      AN    OV;
      =     L      0.0;
      A     L      0.0;
      A(    ;
      A     M   1014.1;
      A(    ;
      A     I   1010.3;
      A(    ;
      ON    I     68.7;
      ON    I     69.4;
      )     ;
      O     ;
      A     I   1018.2;
      A(    ;
      ON    I     68.3;
      ON    I     69.2;
      )     ;
      )     ;
      O     ;
      A     M   1014.0;
      A(    ;
      O     I   1018.2;
      O     ;
      A     I   1018.3;
      A     M    284.0;
      A     M   4710.0;
      )     ;
      A(    ;
      ON    I     71.3;
      ON    I     71.4;
      )     ;
      )     ;
      =     L      0.1;
      A     L      0.1;
      A     T     12;
      S     M   1003.2;
      A     L      0.1;
      AN    M   1004.0;
      AN    M   1004.1;
      AN    M   6060.1;
      AN    M   6260.0;
      AN    M   6280.0;
      AN    M   1004.2;
      L     S5T#500MS;
      SD    T     12;
      A     L      0.0;
      A     I      0.1;
      A(    ;
      A     M   1014.1;
      A(    ;
      A     I     68.7;
      A     I     69.4;
      A     I     68.3;
      A     I     69.2;
      O     ;
      AN    M   1001.4;
      A     M   1001.6;
      A     I     68.3;
      A     I     69.2;
      )     ;
      O     ;
      A     M   1014.0;
      A     M   1001.6;
      A     I     71.3;
      A     I     71.4;
      )     ;
      R     M   1003.2;
NETWORK
TITLE =
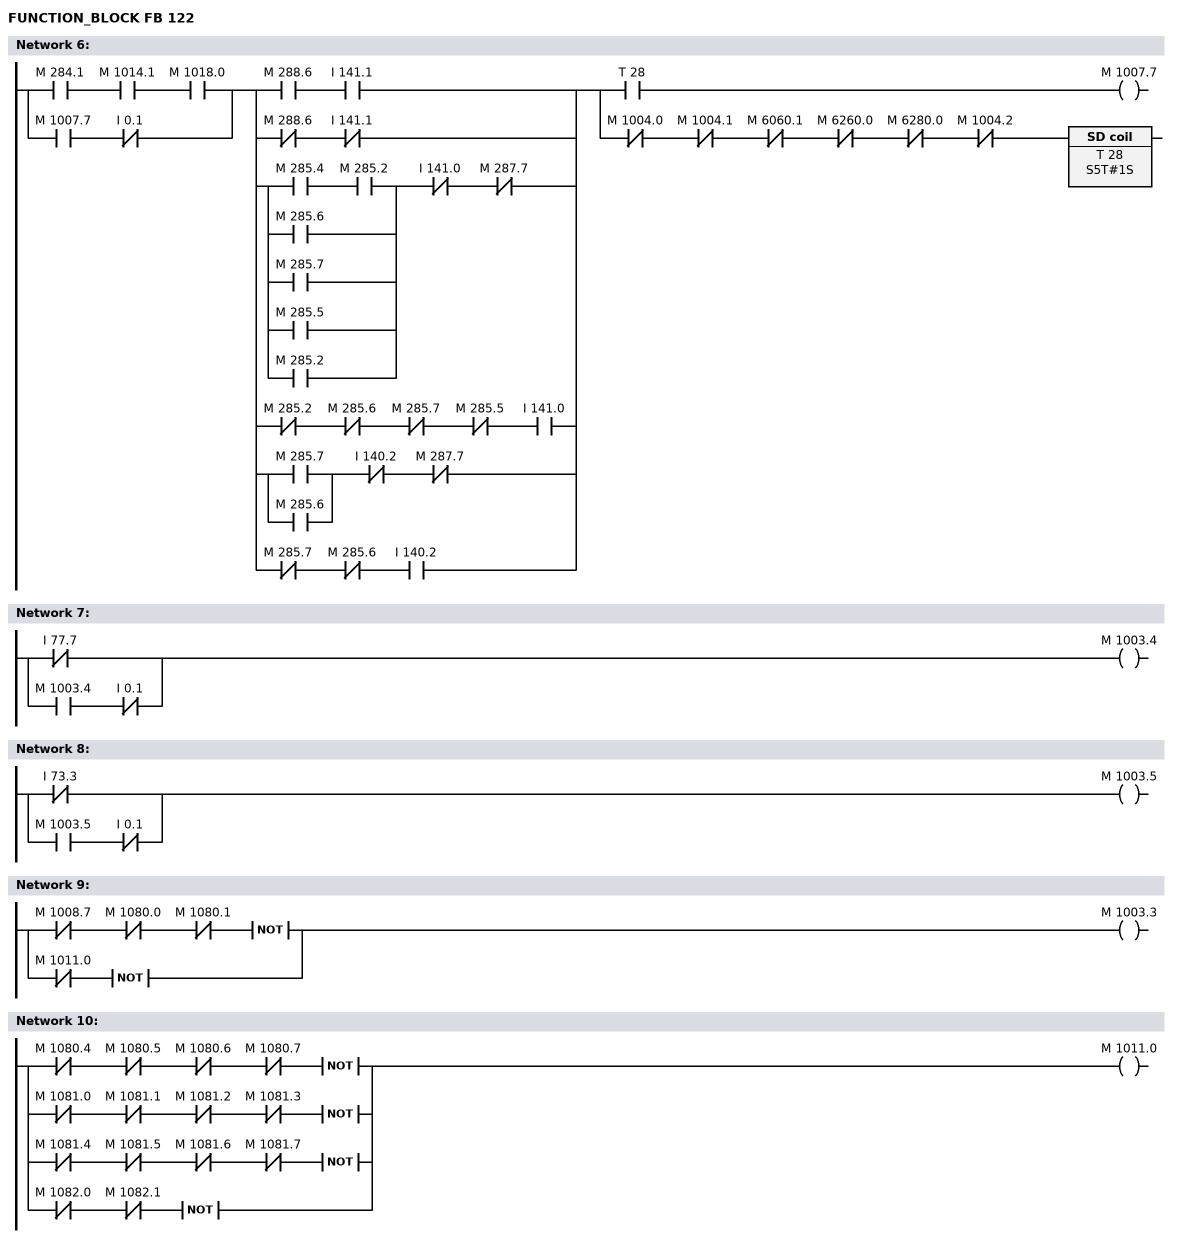

      A(    ;
      A     M    284.1;
      A     M   1014.1;
      A     M   1018.0;
      O     ;
      A     M   1007.7;
      AN    I      0.1;
      )     ;
      A(    ;
      A     M    288.6;
      A     I    141.1;
      O     ;
      AN    M    288.6;
      AN    I    141.1;
      O     ;
      A(    ;
      A     M    285.4;
      A     M    285.2;
      O     M    285.6;
      O     M    285.7;
      O     M    285.5;
      O     M    285.2;
      )     ;
      AN    I    141.0;
      AN    M    287.7;
      O     ;
      AN    M    285.2;
      AN    M    285.6;
      AN    M    285.7;
      AN    M    285.5;
      A     I    141.0;
      O     ;
      A(    ;
      O     M    285.7;
      O     M    285.6;
      )     ;
      AN    I    140.2;
      AN    M    287.7;
      O     ;
      AN    M    285.7;
      AN    M    285.6;
      A     I    140.2;
      )     ;
      =     L      0.0;
      A     L      0.0;
      A     T     28;
      =     M   1007.7;
      A     L      0.0;
      AN    M   1004.0;
      AN    M   1004.1;
      AN    M   6060.1;
      AN    M   6260.0;
      AN    M   6280.0;
      AN    M   1004.2;
      L     S5T#1S;
      SD    T     28;
NETWORK
TITLE =

      ON    I     77.7;
      O     ;
      A     M   1003.4;
      AN    I      0.1;
      =     M   1003.4;
NETWORK
TITLE =

      ON    I     73.3;
      O     ;
      A     M   1003.5;
      AN    I      0.1;
      =     M   1003.5;
NETWORK
TITLE =

      AN    M   1008.7;
      AN    M   1080.0;
      AN    M   1080.1;
      NOT   ;
      O(    ;
      AN    M   1011.0;
      NOT   ;
      )     ;
      =     M   1003.3;
NETWORK
TITLE =

      AN    M   1080.4;
      AN    M   1080.5;
      AN    M   1080.6;
      AN    M   1080.7;
      NOT   ;
      O(    ;
      AN    M   1081.0;
      AN    M   1081.1;
      AN    M   1081.2;
      AN    M   1081.3;
      NOT   ;
      )     ;
      O(    ;
      AN    M   1081.4;
      AN    M   1081.5;
      AN    M   1081.6;
      AN    M   1081.7;
      NOT   ;
      )     ;
      O(    ;
      AN    M   1082.0;
      AN    M   1082.1;
      NOT   ;
      )     ;
      =     M   1011.0;
NETWORK
TITLE =

      AN    OV;
      =     L      0.0;
      A     L      0.0;
      A(    ;
      A     M   1000.6;
      A     I   1016.0;
      AN    M   1001.5;
      AN    M   1001.6;
      A(    ;
      A     DB100.DBX   44.1;
      A     M    264.1;
      A(    ;
      A     DB100.DBX   48.4;
      A     M    268.5;
      O     ;
      A     DB100.DBX   48.5;
      A     M    268.4;
      )     ;
      O     ;
      A     DB100.DBX   44.1;
      A     M    264.0;
      O     ;
      A     DB100.DBX   44.0;
      A     M    264.1;
      O     ;
      A(    ;
      L     MD   260;
      L     DB100.DBD   40;
      <>I   ;
      )     ;
      A     M   1011.6;
      A     M    505.0;
      )     ;
      O     M   1003.0;
      )     ;
      AN    I      0.1;
      AN    M   1004.0;
      AN    M   1004.1;
      AN    M   6060.1;
      AN    M   6260.0;
      AN    M   6280.0;
      AN    M   1004.2;
      AN    I    101.0;
      =     M   1003.0;
      A     L      0.0;
      A     I   1018.5;
      S     M   1001.5;
      A     L      0.0;
      A     I   1016.0;
      R     M   1001.5;
NETWORK
TITLE =
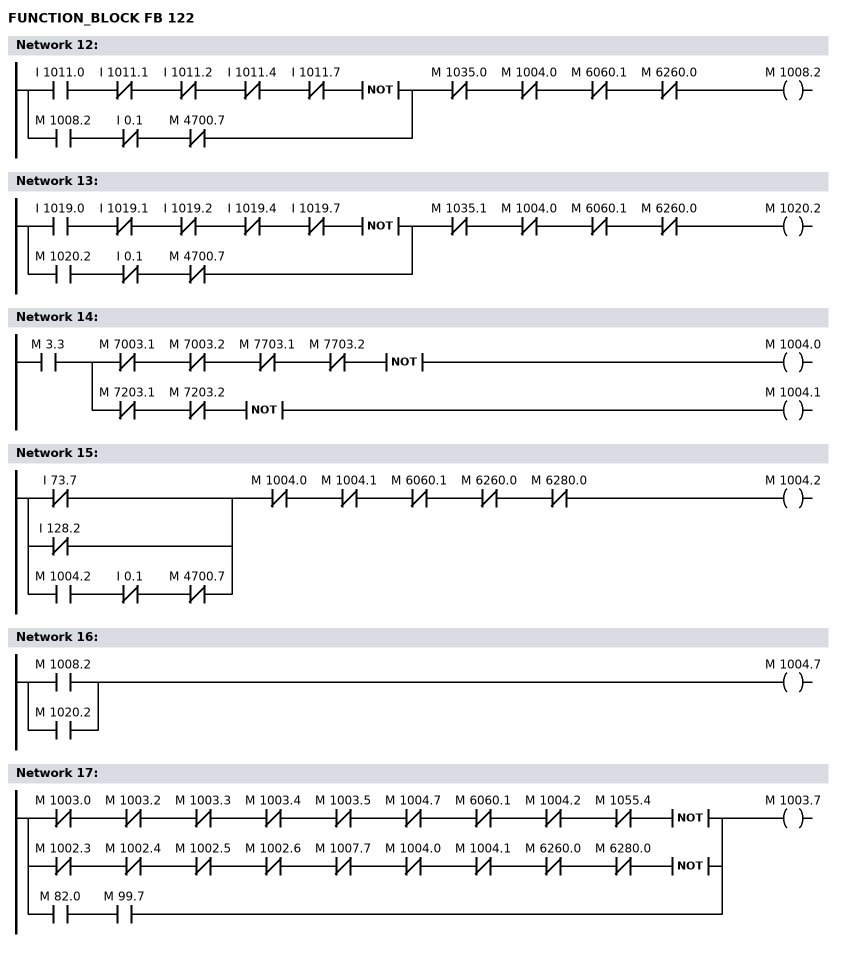

      A(    ;
      A     I   1011.0;
      AN    I   1011.1;
      AN    I   1011.2;
      AN    I   1011.4;
      AN    I   1011.7;
      NOT   ;
      O     ;
      A     M   1008.2;
      AN    I      0.1;
      AN    M   4700.7;
      )     ;
      AN    M   1035.0;
      AN    M   1004.0;
      AN    M   6060.1;
      AN    M   6260.0;
      =     M   1008.2;
NETWORK
TITLE =

      A(    ;
      A     I   1019.0;
      AN    I   1019.1;
      AN    I   1019.2;
      AN    I   1019.4;
      AN    I   1019.7;
      NOT   ;
      O     ;
      A     M   1020.2;
      AN    I      0.1;
      AN    M   4700.7;
      )     ;
      AN    M   1035.1;
      AN    M   1004.0;
      AN    M   6060.1;
      AN    M   6260.0;
      =     M   1020.2;
NETWORK
TITLE =

      A     M      3.3;
      =     L      0.0;
      A     L      0.0;
      AN    M   7003.1;
      AN    M   7003.2;
      AN    M   7703.1;
      AN    M   7703.2;
      NOT   ;
      =     M   1004.0;
      A     L      0.0;
      AN    M   7203.1;
      AN    M   7203.2;
      NOT   ;
      =     M   1004.1;
NETWORK
TITLE =

      A(    ;
      ON    I     73.7;
      ON    I    128.2;
      O     ;
      A     M   1004.2;
      AN    I      0.1;
      AN    M   4700.7;
      )     ;
      AN    M   1004.0;
      AN    M   1004.1;
      AN    M   6060.1;
      AN    M   6260.0;
      AN    M   6280.0;
      =     M   1004.2;
NETWORK
TITLE =

      O     M   1008.2;
      O     M   1020.2;
      =     M   1004.7;
NETWORK
TITLE =

      AN    M   1003.0;
      AN    M   1003.2;
      AN    M   1003.3;
      AN    M   1003.4;
      AN    M   1003.5;
      AN    M   1004.7;
      AN    M   6060.1;
      AN    M   1004.2;
      AN    M   1055.4;
      NOT   ;
      O(    ;
      AN    M   1002.3;
      AN    M   1002.4;
      AN    M   1002.5;
      AN    M   1002.6;
      AN    M   1007.7;
      AN    M   1004.0;
      AN    M   1004.1;
      AN    M   6260.0;
      AN    M   6280.0;
      NOT   ;
      )     ;
      O     ;
      A     M     82.0;
      A     M     99.7;
      =     M   1003.7;
END_FUNCTION_BLOCK

DATA_BLOCK DB 122
TITLE =
VERSION : 0.0

 FB 122
BEGIN
END_DATA_BLOCK

FUNCTION FC 122 : VOID
TITLE =
VERSION : 0.1

BEGIN
NETWORK
TITLE =
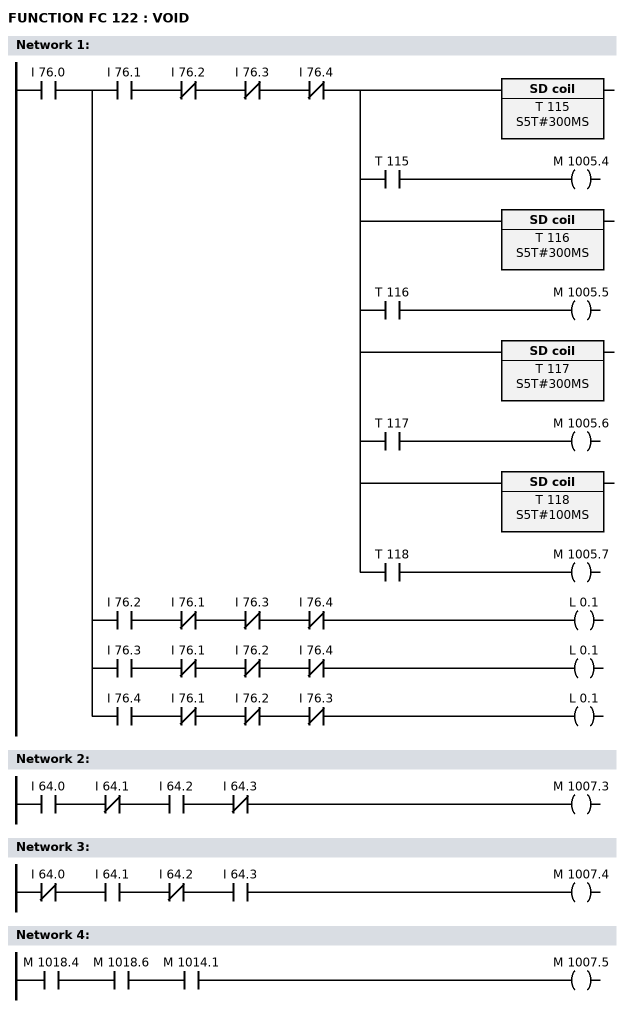

      A     I     76.0;
      =     L      0.0;
      A     L      0.0;
      A     I     76.1;
      AN    I     76.2;
      AN    I     76.3;
      AN    I     76.4;
      =     L      0.1;
      A     L      0.1;
      BLD   102;
      L     S5T#300MS;
      SD    T    115;
      A     L      0.1;
      A     T    115;
      =     M   1005.4;
      A     L      0.0;
      A     I     76.2;
      AN    I     76.1;
      AN    I     76.3;
      AN    I     76.4;
      =     L      0.1;
      A     L      0.1;
      BLD   102;
      L     S5T#300MS;
      SD    T    116;
      A     L      0.1;
      A     T    116;
      =     M   1005.5;
      A     L      0.0;
      A     I     76.3;
      AN    I     76.1;
      AN    I     76.2;
      AN    I     76.4;
      =     L      0.1;
      A     L      0.1;
      BLD   102;
      L     S5T#300MS;
      SD    T    117;
      A     L      0.1;
      A     T    117;
      =     M   1005.6;
      A     L      0.0;
      A     I     76.4;
      AN    I     76.1;
      AN    I     76.2;
      AN    I     76.3;
      =     L      0.1;
      A     L      0.1;
      BLD   102;
      L     S5T#100MS;
      SD    T    118;
      A     L      0.1;
      A     T    118;
      =     M   1005.7;
NETWORK
TITLE =

      A     I     64.0;
      AN    I     64.1;
      A     I     64.2;
      AN    I     64.3;
      =     M   1007.3;
NETWORK
TITLE =

      AN    I     64.0;
      A     I     64.1;
      AN    I     64.2;
      A     I     64.3;
      =     M   1007.4;
NETWORK
TITLE =

      A     M   1018.4;
      A     M   1018.6;
      A     M   1014.1;
      =     M   1007.5;
NETWORK
TITLE =

NETWORK
TITLE =

      AN    OV;
      =     L      0.0;
      A     L      0.0;
      A     I     64.6;
      AN    I     64.7;
      =     M   1012.0;
      A     L      0.0;
      AN    I     64.6;
      A     I     64.7;
      =     M   1012.1;
      A     L      0.0;
      A     I     70.6;
      AN    I     70.7;
      A     I     71.0;
      AN    I     71.1;
      =     M   1012.4;
      A     L      0.0;
      AN    I     70.6;
      A     I     70.7;
      AN    I     71.0;
      A     I     71.1;
      =     M   1012.5;
NETWORK
TITLE =

      AN    OV;
      =     L      0.0;
      A     L      0.0;
      A     I     65.0;
      AN    I     65.1;
      A     I     65.2;
      AN    I     65.3;
      A     I     65.4;
      AN    I     65.5;
      A     I     65.6;
      AN    I     65.7;
      A     I     68.1;
      AN    I     68.2;
      A     I     64.4;
      AN    I     64.5;
      A     I     68.4;
      AN    I     68.5;
      A     I     69.0;
      AN    I     69.1;
      A     I     77.0;
      AN    I     77.1;
      =     M   1017.0;
      A     L      0.0;
      AN    I     65.0;
      A     I     65.1;
      AN    I     65.2;
      A     I     65.3;
      AN    I     65.4;
      A     I     65.5;
      AN    I     65.6;
      A     I     65.7;
      AN    I     68.1;
      A     I     68.2;
      AN    I     64.4;
      A     I     64.5;
      AN    I     68.4;
      A     I     68.5;
      AN    I     69.0;
      A     I     69.1;
      AN    I     77.0;
      A(    ;
      O     I     77.1;
      ON    I     77.0;
      )     ;
      =     M   1017.1;
NETWORK
TITLE =

      AN    OV;
      =     L      0.0;
      A     L      0.0;
      A     I     66.5;
      AN    I     67.5;
      =     M   1017.2;
      A     L      0.0;
      AN    I     66.5;
      A     I     67.5;
      =     M   1017.3;
      A     L      0.0;
      A     I     68.0;
      AN    I     68.6;
      A(    ;
      O     I     72.0;
      ON    I     73.2;
      )     ;
      AN    I     73.2;
      =     M   1017.4;
      A     L      0.0;
      AN    I     68.0;
      A     I     68.6;
      AN    I     72.0;
      A     I     73.2;
      =     M   1017.5;
NETWORK
TITLE =

      AN    OV;
      =     L      0.0;
      A     L      0.0;
      A     I    140.0;
      AN    I    140.1;
      =     M   1018.0;
      A     L      0.0;
      AN    I    140.0;
      A     I    140.1;
      =     M   1018.1;
      A     L      0.0;
      A     I    140.6;
      AN    I    140.7;
      =     M   1018.2;
      A     L      0.0;
      AN    I    140.6;
      A     I    140.7;
      =     M   1018.3;
NETWORK
TITLE =

      AN    OV;
      =     L      0.0;
      A     L      0.0;
      A     M   1017.2;
      A     M   1018.0;
      =     M   1018.4;
      A     L      0.0;
      A     M   1017.3;
      A     M   1018.1;
      =     M   1018.5;
      A     L      0.0;
      A     M   1017.4;
      A     M   1018.2;
      =     M   1018.6;
      A     L      0.0;
      A     M   1017.5;
      A     M   1018.3;
      =     M   1018.7;
      A     L      0.0;
      A     M   1007.3;
      A     M   1005.4;
      =     L      0.1;
      A     L      0.1;
      A     M   1017.0;
      A     M   1012.1;
      A     M   1012.5;
      =     M   1014.1;
      A     L      0.1;
      A     M   1012.0;
      A     M   1017.1;
      A     M   1012.4;
      =     M   1014.0;
NETWORK
TITLE =

NETWORK
TITLE =
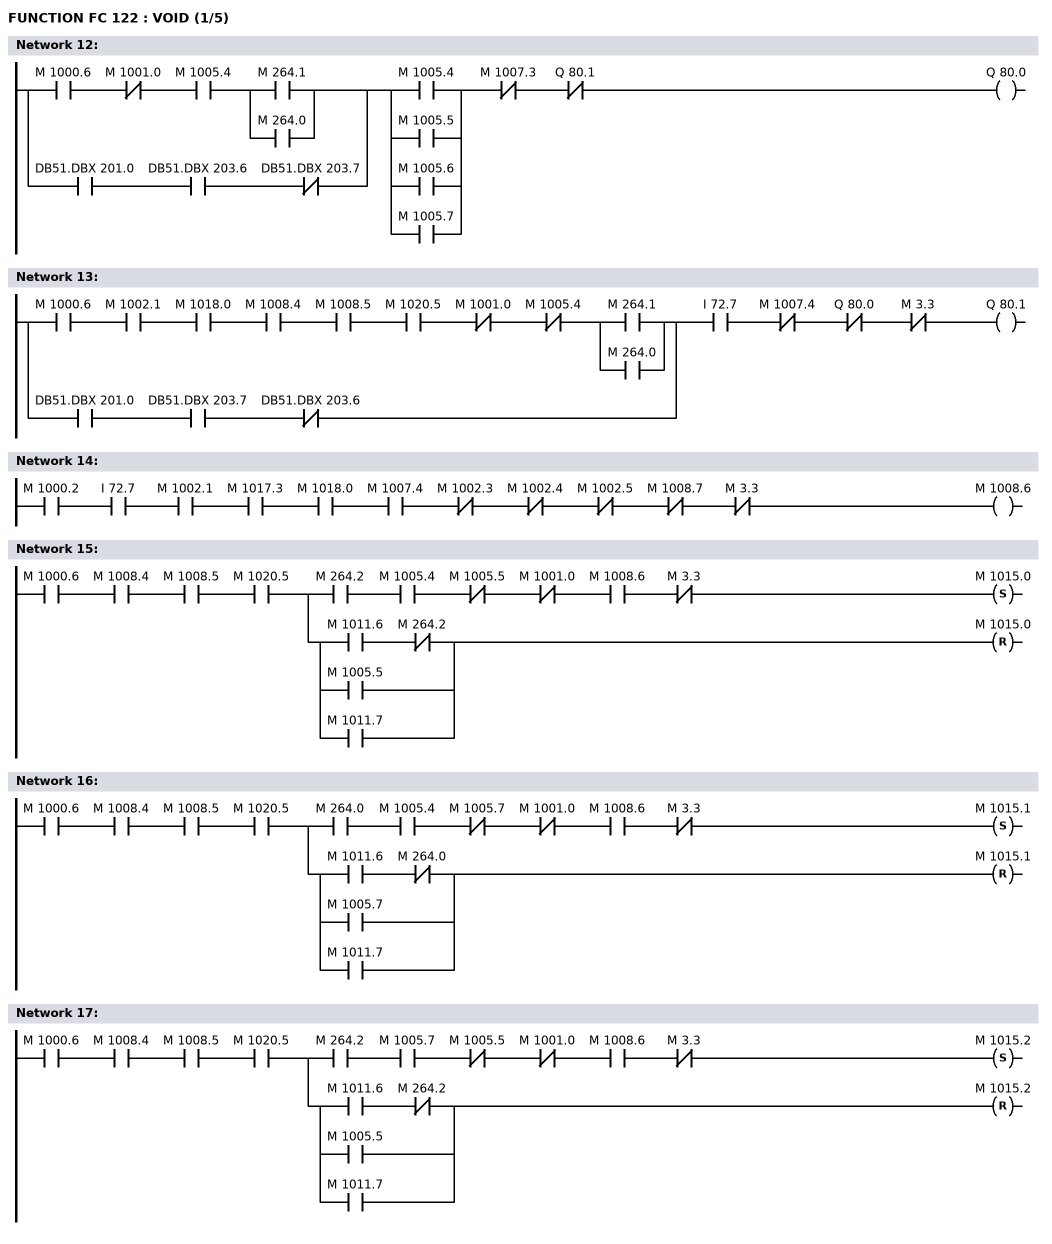

      A(    ;
      A     M   1000.6;
      AN    M   1001.0;
      A     M   1005.4;
      A(    ;
      O     M    264.1;
      O     M    264.0;
      )     ;
      O     ;
      A     DB51.DBX  201.0;
      A     DB51.DBX  203.6;
      AN    DB51.DBX  203.7;
      )     ;
      A(    ;
      O     M   1005.4;
      O     M   1005.5;
      O     M   1005.6;
      O     M   1005.7;
      )     ;
      AN    M   1007.3;
      AN    Q     80.1;
      =     Q     80.0;
NETWORK
TITLE =

      A(    ;
      A     M   1000.6;
      A     M   1002.1;
      A     M   1018.0;
      A     M   1008.4;
      A     M   1008.5;
      A     M   1020.5;
      AN    M   1001.0;
      AN    M   1005.4;
      A(    ;
      O     M    264.1;
      O     M    264.0;
      )     ;
      O     ;
      A     DB51.DBX  201.0;
      A     DB51.DBX  203.7;
      AN    DB51.DBX  203.6;
      )     ;
      A     I     72.7;
      AN    M   1007.4;
      AN    Q     80.0;
      AN    M      3.3;
      =     Q     80.1;
NETWORK
TITLE =

      A     M   1000.2;
      A     I     72.7;
      A     M   1002.1;
      A     M   1017.3;
      A     M   1018.0;
      A     M   1007.4;
      AN    M   1002.3;
      AN    M   1002.4;
      AN    M   1002.5;
      AN    M   1008.7;
      AN    M      3.3;
      =     M   1008.6;
NETWORK
TITLE =

      A     M   1000.6;
      A     M   1008.4;
      A     M   1008.5;
      A     M   1020.5;
      =     L      0.0;
      A     L      0.0;
      A     M    264.2;
      A     M   1005.4;
      AN    M   1005.5;
      AN    M   1001.0;
      A     M   1008.6;
      AN    M      3.3;
      S     M   1015.0;
      A     L      0.0;
      A(    ;
      A     M   1011.6;
      AN    M    264.2;
      O     M   1005.5;
      O     M   1011.7;
      )     ;
      R     M   1015.0;
NETWORK
TITLE =

      A     M   1000.6;
      A     M   1008.4;
      A     M   1008.5;
      A     M   1020.5;
      =     L      0.0;
      A     L      0.0;
      A     M    264.0;
      A     M   1005.4;
      AN    M   1005.7;
      AN    M   1001.0;
      A     M   1008.6;
      AN    M      3.3;
      S     M   1015.1;
      A     L      0.0;
      A(    ;
      A     M   1011.6;
      AN    M    264.0;
      O     M   1005.7;
      O     M   1011.7;
      )     ;
      R     M   1015.1;
NETWORK
TITLE =

      A     M   1000.6;
      A     M   1008.4;
      A     M   1008.5;
      A     M   1020.5;
      =     L      0.0;
      A     L      0.0;
      A     M    264.2;
      A     M   1005.7;
      AN    M   1005.5;
      AN    M   1001.0;
      A     M   1008.6;
      AN    M      3.3;
      S     M   1015.2;
      A     L      0.0;
      A(    ;
      A     M   1011.6;
      AN    M    264.2;
      O     M   1005.5;
      O     M   1011.7;
      )     ;
      R     M   1015.2;
NETWORK
TITLE =
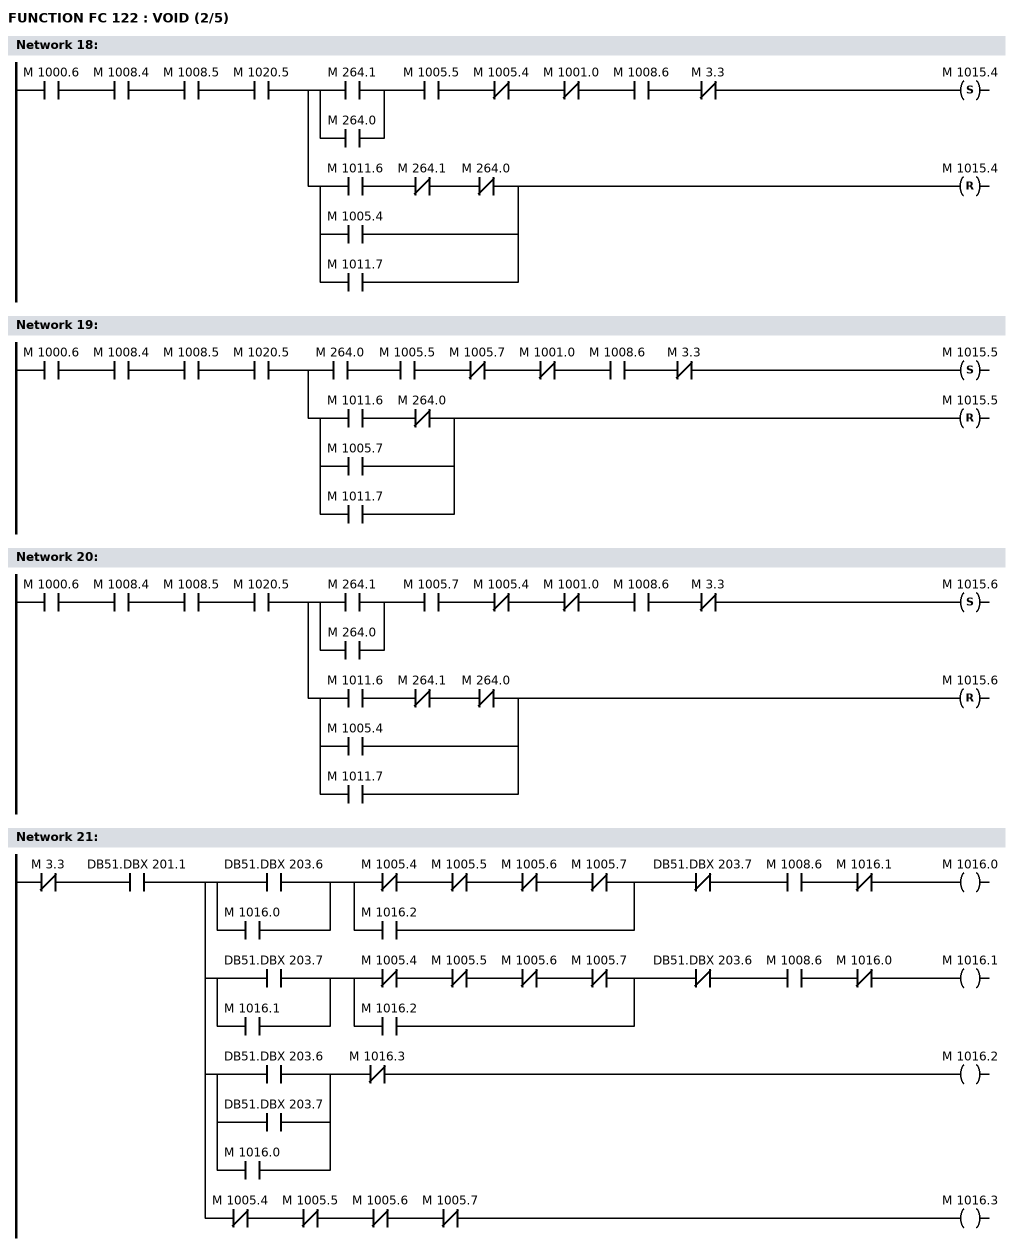

      A     M   1000.6;
      A     M   1008.4;
      A     M   1008.5;
      A     M   1020.5;
      =     L      0.0;
      A     L      0.0;
      A(    ;
      O     M    264.1;
      O     M    264.0;
      )     ;
      A     M   1005.5;
      AN    M   1005.4;
      AN    M   1001.0;
      A     M   1008.6;
      AN    M      3.3;
      S     M   1015.4;
      A     L      0.0;
      A(    ;
      A     M   1011.6;
      AN    M    264.1;
      AN    M    264.0;
      O     M   1005.4;
      O     M   1011.7;
      )     ;
      R     M   1015.4;
NETWORK
TITLE =

      A     M   1000.6;
      A     M   1008.4;
      A     M   1008.5;
      A     M   1020.5;
      =     L      0.0;
      A     L      0.0;
      A     M    264.0;
      A     M   1005.5;
      AN    M   1005.7;
      AN    M   1001.0;
      A     M   1008.6;
      AN    M      3.3;
      S     M   1015.5;
      A     L      0.0;
      A(    ;
      A     M   1011.6;
      AN    M    264.0;
      O     M   1005.7;
      O     M   1011.7;
      )     ;
      R     M   1015.5;
NETWORK
TITLE =

      A     M   1000.6;
      A     M   1008.4;
      A     M   1008.5;
      A     M   1020.5;
      =     L      0.0;
      A     L      0.0;
      A(    ;
      O     M    264.1;
      O     M    264.0;
      )     ;
      A     M   1005.7;
      AN    M   1005.4;
      AN    M   1001.0;
      A     M   1008.6;
      AN    M      3.3;
      S     M   1015.6;
      A     L      0.0;
      A(    ;
      A     M   1011.6;
      AN    M    264.1;
      AN    M    264.0;
      O     M   1005.4;
      O     M   1011.7;
      )     ;
      R     M   1015.6;
NETWORK
TITLE =

      AN    M      3.3;
      A     DB51.DBX  201.1;
      =     L      0.0;
      A     L      0.0;
      A(    ;
      O     DB51.DBX  203.6;
      O     M   1016.0;
      )     ;
      A(    ;
      AN    M   1005.4;
      AN    M   1005.5;
      AN    M   1005.6;
      AN    M   1005.7;
      O     M   1016.2;
      )     ;
      AN    DB51.DBX  203.7;
      A     M   1008.6;
      AN    M   1016.1;
      =     M   1016.0;
      A     L      0.0;
      A(    ;
      O     DB51.DBX  203.7;
      O     M   1016.1;
      )     ;
      A(    ;
      AN    M   1005.4;
      AN    M   1005.5;
      AN    M   1005.6;
      AN    M   1005.7;
      O     M   1016.2;
      )     ;
      AN    DB51.DBX  203.6;
      A     M   1008.6;
      AN    M   1016.0;
      =     M   1016.1;
      A     L      0.0;
      A(    ;
      O     DB51.DBX  203.6;
      O     DB51.DBX  203.7;
      O     M   1016.0;
      )     ;
      AN    M   1016.3;
      =     M   1016.2;
      A     L      0.0;
      AN    M   1005.4;
      AN    M   1005.5;
      AN    M   1005.6;
      AN    M   1005.7;
      =     M   1016.3;
NETWORK
TITLE =
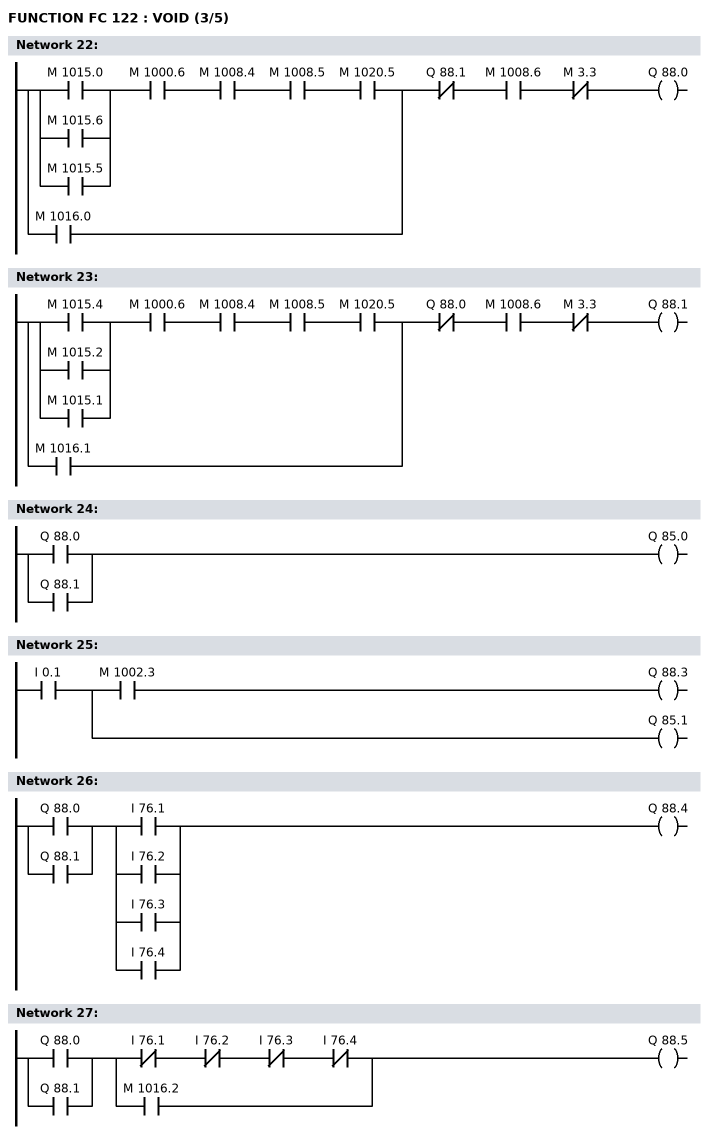

      A(    ;
      A(    ;
      O     M   1015.0;
      O     M   1015.6;
      O     M   1015.5;
      )     ;
      A     M   1000.6;
      A     M   1008.4;
      A     M   1008.5;
      A     M   1020.5;
      O     M   1016.0;
      )     ;
      AN    Q     88.1;
      A     M   1008.6;
      AN    M      3.3;
      =     Q     88.0;
NETWORK
TITLE =

      A(    ;
      A(    ;
      O     M   1015.4;
      O     M   1015.2;
      O     M   1015.1;
      )     ;
      A     M   1000.6;
      A     M   1008.4;
      A     M   1008.5;
      A     M   1020.5;
      O     M   1016.1;
      )     ;
      AN    Q     88.0;
      A     M   1008.6;
      AN    M      3.3;
      =     Q     88.1;
NETWORK
TITLE =

      O     Q     88.0;
      O     Q     88.1;
      =     Q     85.0;
NETWORK
TITLE =

      A     I      0.1;
      =     L      0.0;
      A     L      0.0;
      A     M   1002.3;
      =     Q     88.3;
      A     L      0.0;
      BLD   102;
      =     Q     85.1;
NETWORK
TITLE =

      A(    ;
      O     Q     88.0;
      O     Q     88.1;
      )     ;
      A(    ;
      O     I     76.1;
      O     I     76.2;
      O     I     76.3;
      O     I     76.4;
      )     ;
      =     Q     88.4;
NETWORK
TITLE =

      A(    ;
      O     Q     88.0;
      O     Q     88.1;
      )     ;
      A(    ;
      AN    I     76.1;
      AN    I     76.2;
      AN    I     76.3;
      AN    I     76.4;
      O     M   1016.2;
      )     ;
      =     Q     88.5;
NETWORK
TITLE =

NETWORK
TITLE =
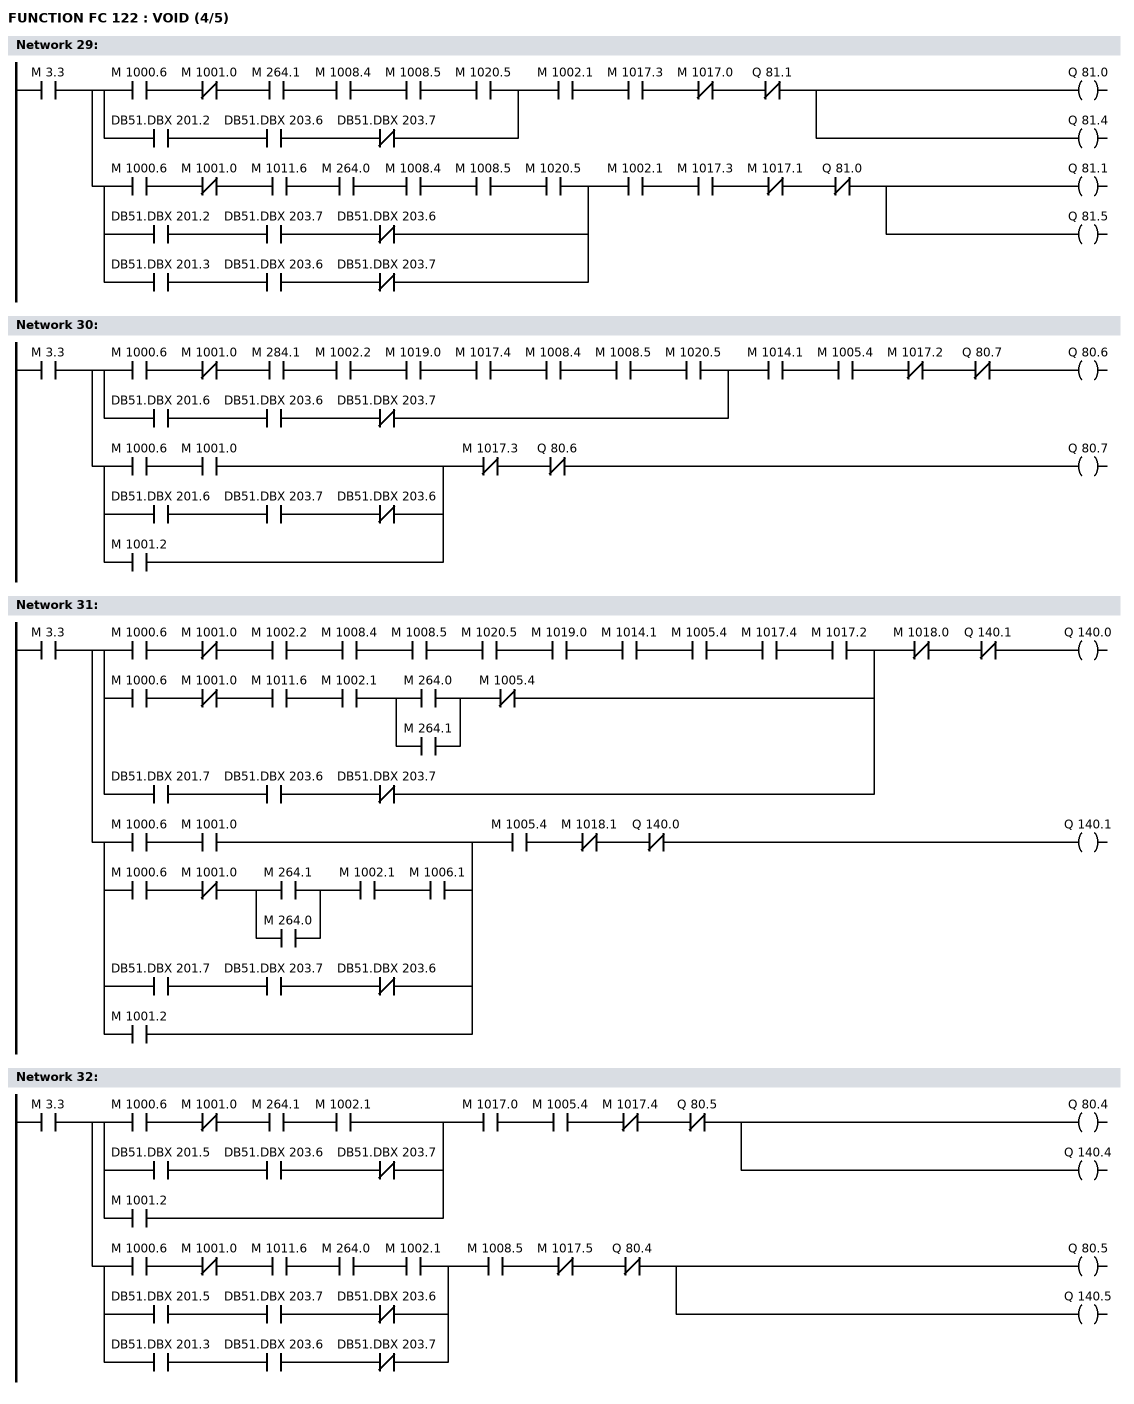

      A     M      3.3;
      =     L      0.0;
      A     L      0.0;
      A(    ;
      A     M   1000.6;
      AN    M   1001.0;
      A     M    264.1;
      A     M   1008.4;
      A     M   1008.5;
      A     M   1020.5;
      O     ;
      A     DB51.DBX  201.2;
      A     DB51.DBX  203.6;
      AN    DB51.DBX  203.7;
      )     ;
      A     M   1002.1;
      A     M   1017.3;
      AN    M   1017.0;
      AN    Q     81.1;
      =     Q     81.0;
      =     Q     81.4;
      A     L      0.0;
      A(    ;
      A     M   1000.6;
      AN    M   1001.0;
      A     M   1011.6;
      A     M    264.0;
      A     M   1008.4;
      A     M   1008.5;
      A     M   1020.5;
      O     ;
      A     DB51.DBX  201.2;
      A     DB51.DBX  203.7;
      AN    DB51.DBX  203.6;
      O     ;
      A     DB51.DBX  201.3;
      A     DB51.DBX  203.6;
      AN    DB51.DBX  203.7;
      )     ;
      A     M   1002.1;
      A     M   1017.3;
      AN    M   1017.1;
      AN    Q     81.0;
      =     Q     81.1;
      =     Q     81.5;
NETWORK
TITLE =

      A     M      3.3;
      =     L      0.0;
      A     L      0.0;
      A(    ;
      A     M   1000.6;
      AN    M   1001.0;
      A     M    284.1;
      A     M   1002.2;
      A     M   1019.0;
      A     M   1017.4;
      A     M   1008.4;
      A     M   1008.5;
      A     M   1020.5;
      O     ;
      A     DB51.DBX  201.6;
      A     DB51.DBX  203.6;
      AN    DB51.DBX  203.7;
      )     ;
      A     M   1014.1;
      A     M   1005.4;
      AN    M   1017.2;
      AN    Q     80.7;
      =     Q     80.6;
      A     L      0.0;
      A(    ;
      A     M   1000.6;
      A     M   1001.0;
      O     ;
      A     DB51.DBX  201.6;
      A     DB51.DBX  203.7;
      AN    DB51.DBX  203.6;
      O     M   1001.2;
      )     ;
      AN    M   1017.3;
      AN    Q     80.6;
      =     Q     80.7;
NETWORK
TITLE =

      A     M      3.3;
      =     L      0.0;
      A     L      0.0;
      A(    ;
      A     M   1000.6;
      AN    M   1001.0;
      A     M   1002.2;
      A     M   1008.4;
      A     M   1008.5;
      A     M   1020.5;
      A     M   1019.0;
      A     M   1014.1;
      A     M   1005.4;
      A     M   1017.4;
      A     M   1017.2;
      O     ;
      A     M   1000.6;
      AN    M   1001.0;
      A     M   1011.6;
      A     M   1002.1;
      A(    ;
      O     M    264.0;
      O     M    264.1;
      )     ;
      AN    M   1005.4;
      O     ;
      A     DB51.DBX  201.7;
      A     DB51.DBX  203.6;
      AN    DB51.DBX  203.7;
      )     ;
      AN    M   1018.0;
      AN    Q    140.1;
      =     Q    140.0;
      A     L      0.0;
      A(    ;
      A     M   1000.6;
      A     M   1001.0;
      O     ;
      A     M   1000.6;
      AN    M   1001.0;
      A(    ;
      O     M    264.1;
      O     M    264.0;
      )     ;
      A     M   1002.1;
      A     M   1006.1;
      O     ;
      A     DB51.DBX  201.7;
      A     DB51.DBX  203.7;
      AN    DB51.DBX  203.6;
      O     M   1001.2;
      )     ;
      A     M   1005.4;
      AN    M   1018.1;
      AN    Q    140.0;
      =     Q    140.1;
NETWORK
TITLE =

      A     M      3.3;
      =     L      0.0;
      A     L      0.0;
      A(    ;
      A     M   1000.6;
      AN    M   1001.0;
      A     M    264.1;
      A     M   1002.1;
      O     ;
      A     DB51.DBX  201.5;
      A     DB51.DBX  203.6;
      AN    DB51.DBX  203.7;
      O     M   1001.2;
      )     ;
      A     M   1017.0;
      A     M   1005.4;
      AN    M   1017.4;
      AN    Q     80.5;
      =     Q     80.4;
      =     Q    140.4;
      A     L      0.0;
      A(    ;
      A     M   1000.6;
      AN    M   1001.0;
      A     M   1011.6;
      A     M    264.0;
      A     M   1002.1;
      O     ;
      A     DB51.DBX  201.5;
      A     DB51.DBX  203.7;
      AN    DB51.DBX  203.6;
      O     ;
      A     DB51.DBX  201.3;
      A     DB51.DBX  203.6;
      AN    DB51.DBX  203.7;
      )     ;
      A     M   1008.5;
      AN    M   1017.5;
      AN    Q     80.4;
      =     Q     80.5;
      =     Q    140.5;
NETWORK
TITLE =
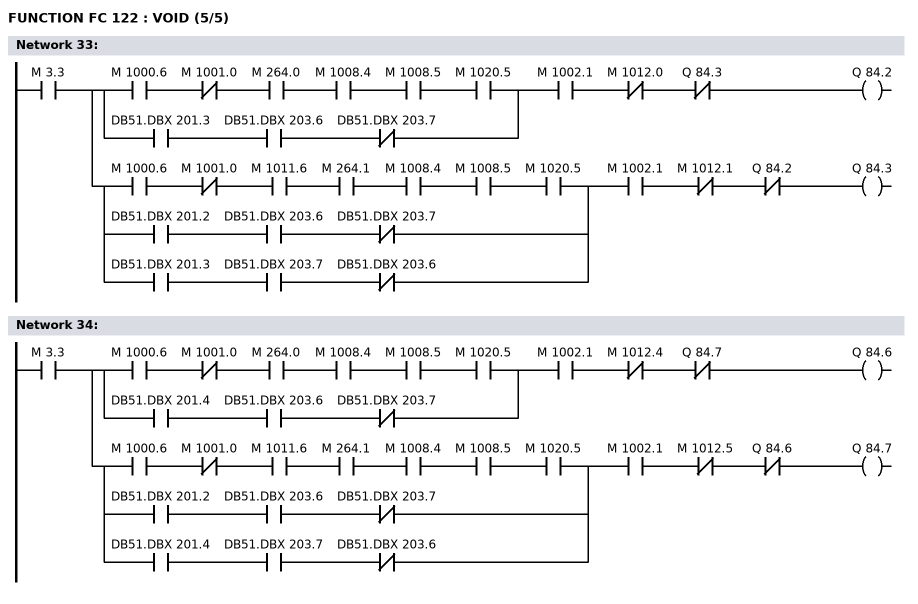

      A     M      3.3;
      =     L      0.0;
      A     L      0.0;
      A(    ;
      A     M   1000.6;
      AN    M   1001.0;
      A     M    264.0;
      A     M   1008.4;
      A     M   1008.5;
      A     M   1020.5;
      O     ;
      A     DB51.DBX  201.3;
      A     DB51.DBX  203.6;
      AN    DB51.DBX  203.7;
      )     ;
      A     M   1002.1;
      AN    M   1012.0;
      AN    Q     84.3;
      =     Q     84.2;
      A     L      0.0;
      A(    ;
      A     M   1000.6;
      AN    M   1001.0;
      A     M   1011.6;
      A     M    264.1;
      A     M   1008.4;
      A     M   1008.5;
      A     M   1020.5;
      O     ;
      A     DB51.DBX  201.2;
      A     DB51.DBX  203.6;
      AN    DB51.DBX  203.7;
      O     ;
      A     DB51.DBX  201.3;
      A     DB51.DBX  203.7;
      AN    DB51.DBX  203.6;
      )     ;
      A     M   1002.1;
      AN    M   1012.1;
      AN    Q     84.2;
      =     Q     84.3;
NETWORK
TITLE =

      A     M      3.3;
      =     L      0.0;
      A     L      0.0;
      A(    ;
      A     M   1000.6;
      AN    M   1001.0;
      A     M    264.0;
      A     M   1008.4;
      A     M   1008.5;
      A     M   1020.5;
      O     ;
      A     DB51.DBX  201.4;
      A     DB51.DBX  203.6;
      AN    DB51.DBX  203.7;
      )     ;
      A     M   1002.1;
      AN    M   1012.4;
      AN    Q     84.7;
      =     Q     84.6;
      A     L      0.0;
      A(    ;
      A     M   1000.6;
      AN    M   1001.0;
      A     M   1011.6;
      A     M    264.1;
      A     M   1008.4;
      A     M   1008.5;
      A     M   1020.5;
      O     ;
      A     DB51.DBX  201.2;
      A     DB51.DBX  203.6;
      AN    DB51.DBX  203.7;
      O     ;
      A     DB51.DBX  201.4;
      A     DB51.DBX  203.7;
      AN    DB51.DBX  203.6;
      )     ;
      A     M   1002.1;
      AN    M   1012.5;
      AN    Q     84.6;
      =     Q     84.7;
END_FUNCTION

FUNCTION FC 123 : VOID
TITLE =
VERSION : 0.1

BEGIN
NETWORK
TITLE =
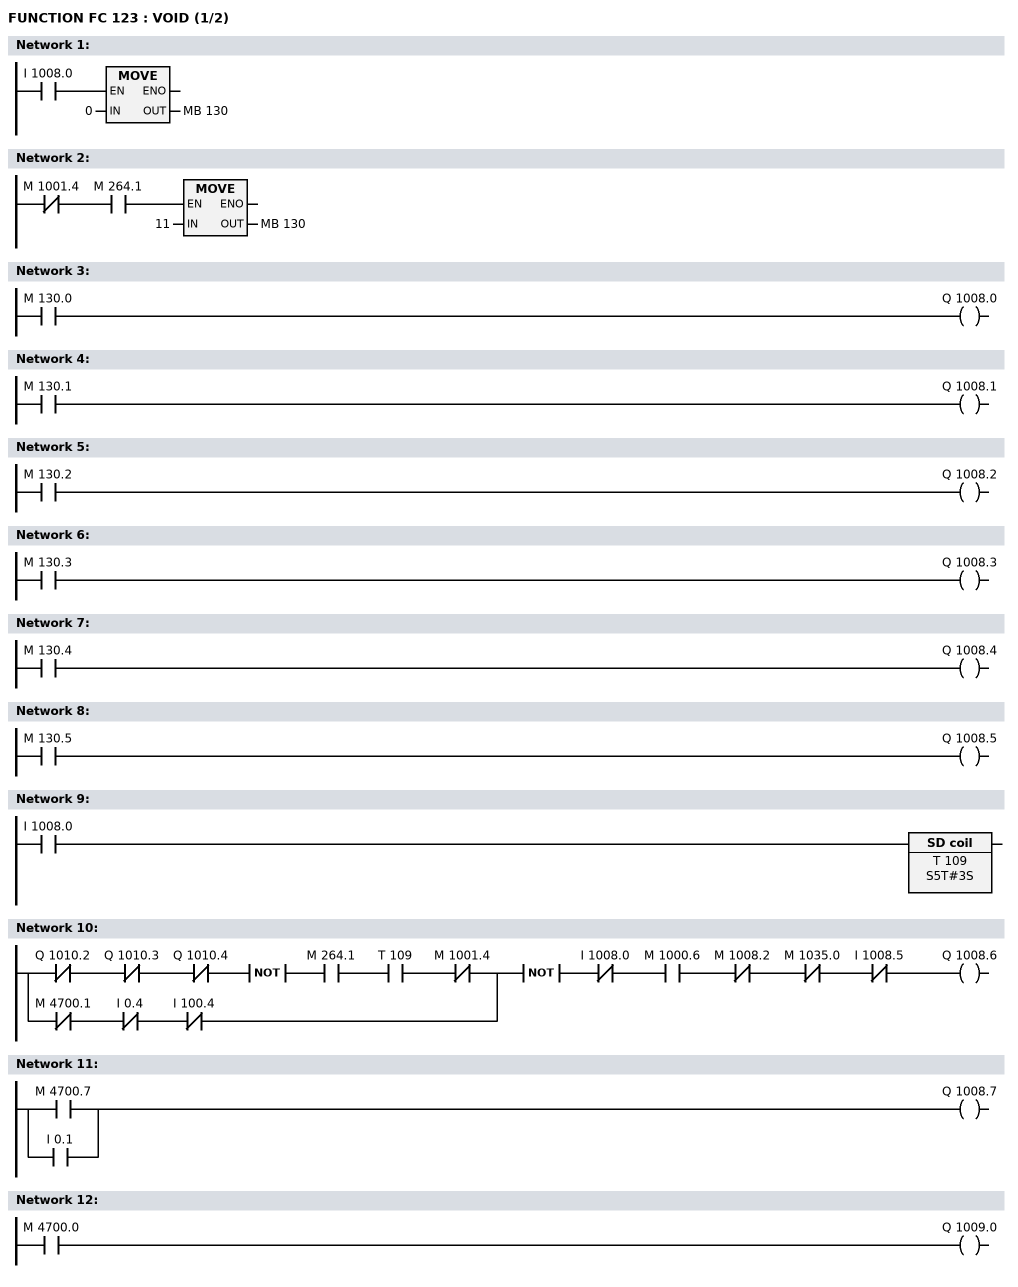

      A     I   1008.0;
      JNB   _001;
      L     0;
      T     MB   130;
_001: NOP   0;
NETWORK
TITLE =

      AN    M   1001.4;
      A     M    264.1;
      JNB   _002;
      L     11;
      T     MB   130;
_002: NOP   0;
NETWORK
TITLE =

      A     M    130.0;
      =     Q   1008.0;
NETWORK
TITLE =

      A     M    130.1;
      =     Q   1008.1;
NETWORK
TITLE =

      A     M    130.2;
      =     Q   1008.2;
NETWORK
TITLE =

      A     M    130.3;
      =     Q   1008.3;
NETWORK
TITLE =

      A     M    130.4;
      =     Q   1008.4;
NETWORK
TITLE =

      A     M    130.5;
      =     Q   1008.5;
NETWORK
TITLE =

      A     I   1008.0;
      L     S5T#3S;
      SD    T    109;
NETWORK
TITLE =

      A(    ;
      AN    Q   1010.2;
      AN    Q   1010.3;
      AN    Q   1010.4;
      NOT   ;
      A     M    264.1;
      A     T    109;
      AN    M   1001.4;
      O     ;
      AN    M   4700.1;
      AN    I      0.4;
      AN    I    100.4;
      NOT   ;
      AN    I   1008.0;
      )     ;
      A     M   1000.6;
      AN    M   1008.2;
      AN    M   1035.0;
      AN    I   1008.5;
      =     Q   1008.6;
NETWORK
TITLE =

      O     M   4700.7;
      O     I      0.1;
      =     Q   1008.7;
NETWORK
TITLE =

      A     M   4700.0;
      =     Q   1009.0;
NETWORK
TITLE =
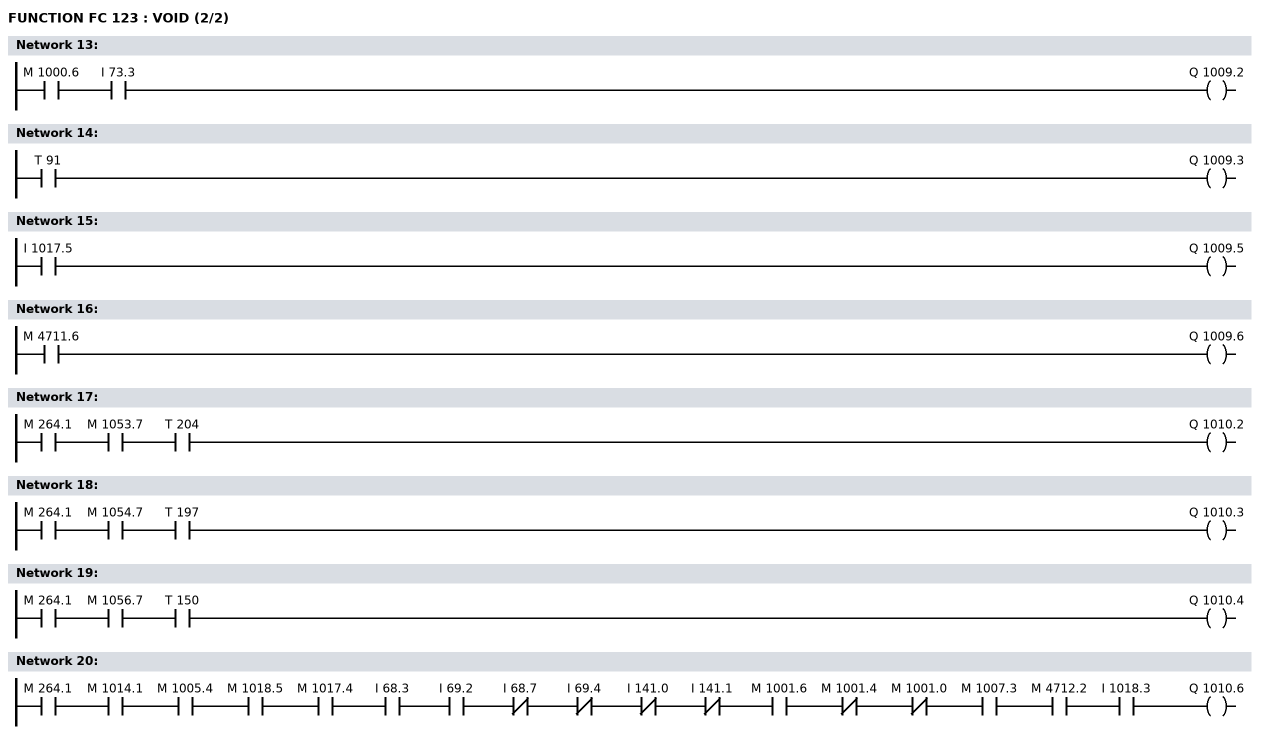

      A     M   1000.6;
      A     I     73.3;
      =     Q   1009.2;
NETWORK
TITLE =

      A     T     91;
      =     Q   1009.3;
NETWORK
TITLE =

      A     I   1017.5;
      =     Q   1009.5;
NETWORK
TITLE =

      A     M   4711.6;
      =     Q   1009.6;
NETWORK
TITLE =

      A     M    264.1;
      A     M   1053.7;
      A     T    204;
      =     Q   1010.2;
NETWORK
TITLE =

      A     M    264.1;
      A     M   1054.7;
      A     T    197;
      =     Q   1010.3;
NETWORK
TITLE =

      A     M    264.1;
      A     M   1056.7;
      A     T    150;
      =     Q   1010.4;
NETWORK
TITLE =

      A     M    264.1;
      A     M   1014.1;
      A     M   1005.4;
      A     M   1018.5;
      A     M   1017.4;
      A     I     68.3;
      A     I     69.2;
      AN    I     68.7;
      AN    I     69.4;
      AN    I    141.0;
      AN    I    141.1;
      A     M   1001.6;
      AN    M   1001.4;
      AN    M   1001.0;
      A     M   1007.3;
      A     M   4712.2;
      A     I   1018.3;
      =     Q   1010.6;
END_FUNCTION

FUNCTION FC 124 : VOID
TITLE =
VERSION : 0.1

BEGIN
NETWORK
TITLE =
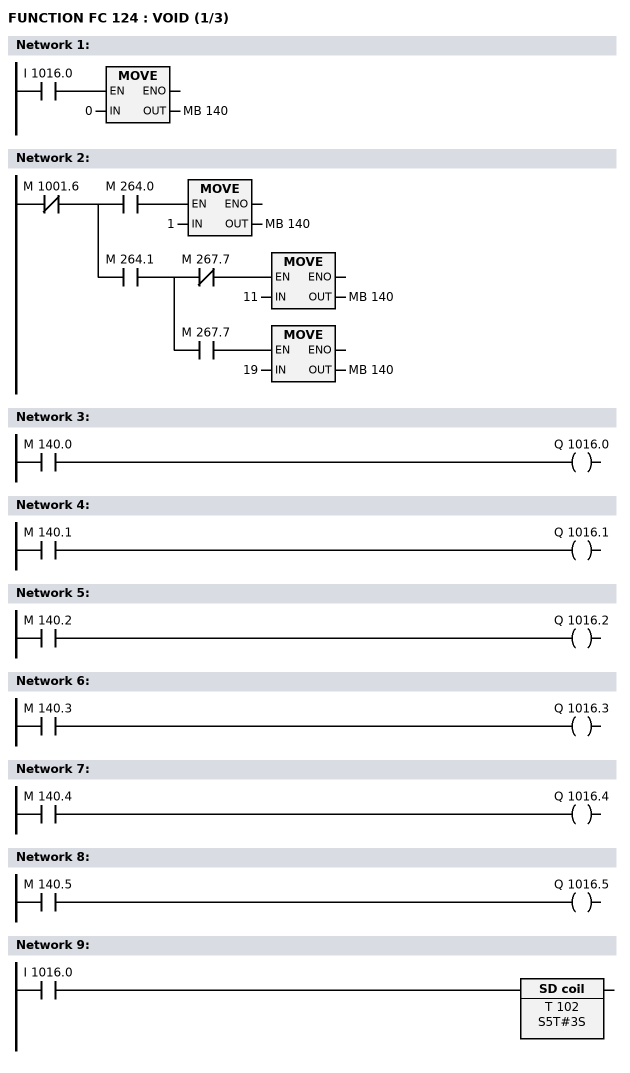

      A     I   1016.0;
      JNB   _001;
      L     0;
      T     MB   140;
_001: NOP   0;
NETWORK
TITLE =

      AN    M   1001.6;
      =     L      0.0;
      A     L      0.0;
      A     M    264.0;
      JNB   _002;
      L     1;
      T     MB   140;
_002: NOP   0;
      A     L      0.0;
      A     M    264.1;
      =     L      0.1;
      A     L      0.1;
      AN    M    267.7;
      JNB   _003;
      L     11;
      T     MB   140;
_003: NOP   0;
      A     L      0.1;
      A     M    267.7;
      JNB   _004;
      L     19;
      T     MB   140;
_004: NOP   0;
NETWORK
TITLE =

      A     M    140.0;
      =     Q   1016.0;
NETWORK
TITLE =

      A     M    140.1;
      =     Q   1016.1;
NETWORK
TITLE =

      A     M    140.2;
      =     Q   1016.2;
NETWORK
TITLE =

      A     M    140.3;
      =     Q   1016.3;
NETWORK
TITLE =

      A     M    140.4;
      =     Q   1016.4;
NETWORK
TITLE =

      A     M    140.5;
      =     Q   1016.5;
NETWORK
TITLE =

      A     I   1016.0;
      L     S5T#3S;
      SD    T    102;
NETWORK
TITLE =
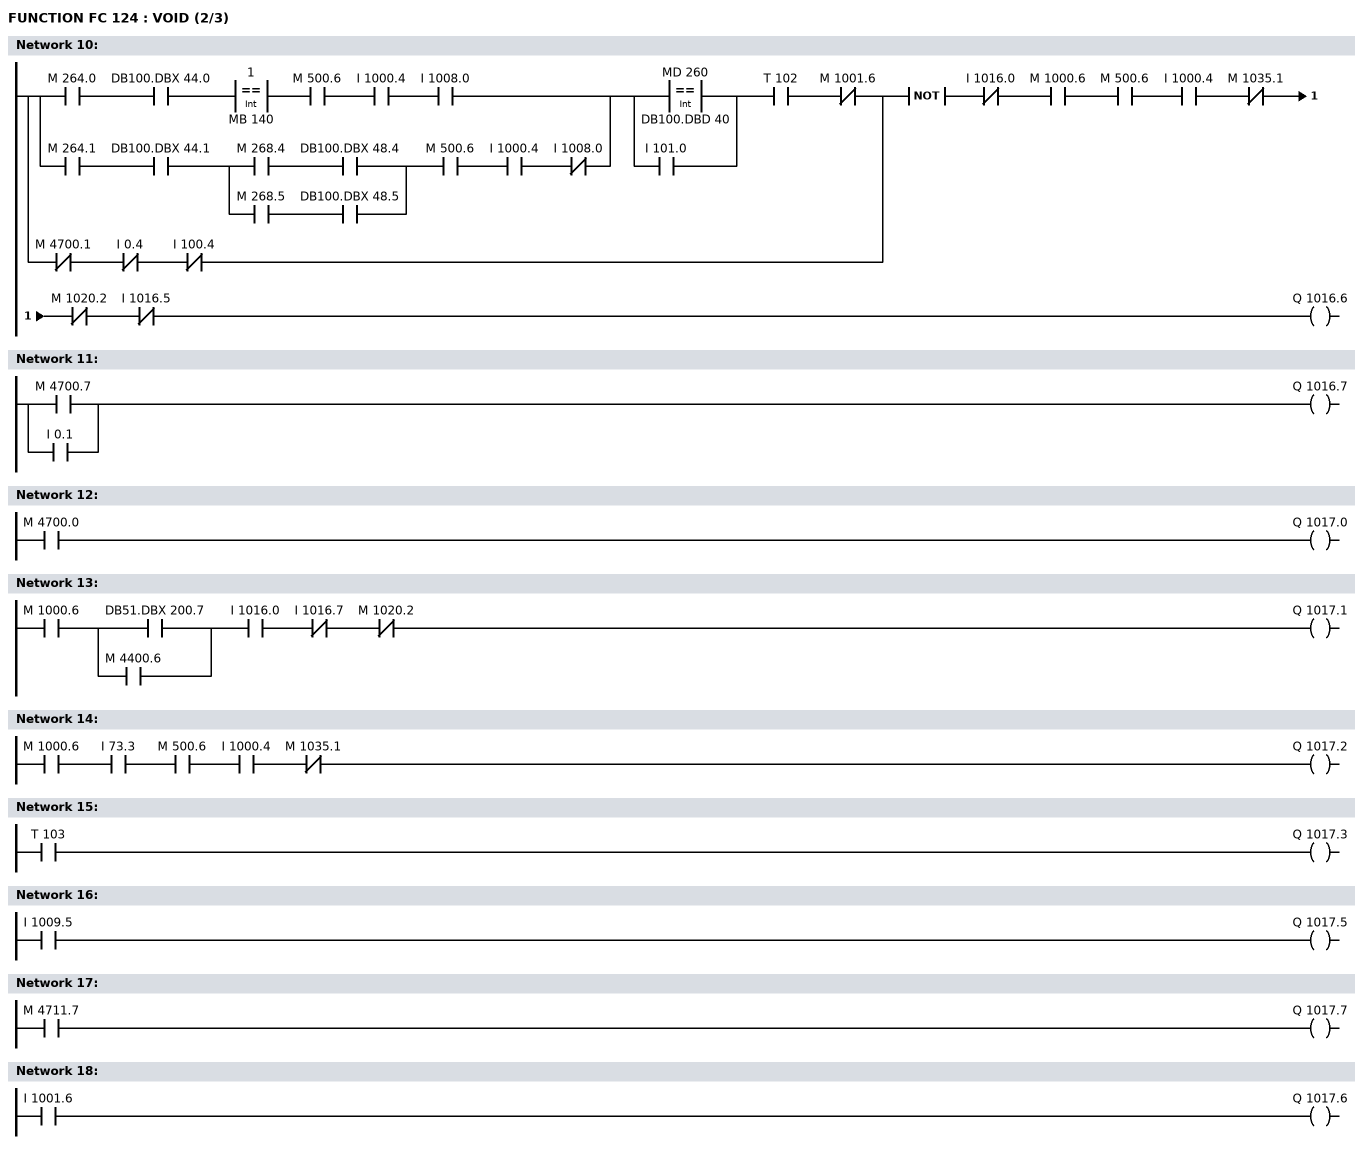

      A(    ;
      A(    ;
      A     M    264.0;
      A     DB100.DBX   44.0;
      A(    ;
      L     1;
      L     MB   140;
      ==I   ;
      )     ;
      A     M    500.6;
      A     I   1000.4;
      A     I   1008.0;
      O     ;
      A     M    264.1;
      A     DB100.DBX   44.1;
      A(    ;
      A     M    268.4;
      A     DB100.DBX   48.4;
      O     ;
      A     M    268.5;
      A     DB100.DBX   48.5;
      )     ;
      A     M    500.6;
      A     I   1000.4;
      AN    I   1008.0;
      )     ;
      A(    ;
      O(    ;
      L     MD   260;
      L     DB100.DBD   40;
      ==I   ;
      )     ;
      O     I    101.0;
      )     ;
      A     T    102;
      AN    M   1001.6;
      O     ;
      AN    M   4700.1;
      AN    I      0.4;
      AN    I    100.4;
      NOT   ;
      AN    I   1016.0;
      )     ;
      A     M   1000.6;
      A     M    500.6;
      A     I   1000.4;
      AN    M   1035.1;
      AN    M   1020.2;
      AN    I   1016.5;
      =     Q   1016.6;
NETWORK
TITLE =

      O     M   4700.7;
      O     I      0.1;
      =     Q   1016.7;
NETWORK
TITLE =

      A     M   4700.0;
      =     Q   1017.0;
NETWORK
TITLE =

      A     M   1000.6;
      A(    ;
      O     DB51.DBX  200.7;
      O     M   4400.6;
      )     ;
      A     I   1016.0;
      AN    I   1016.7;
      AN    M   1020.2;
      =     Q   1017.1;
NETWORK
TITLE =

      A     M   1000.6;
      A     I     73.3;
      A     M    500.6;
      A     I   1000.4;
      AN    M   1035.1;
      =     Q   1017.2;
NETWORK
TITLE =

      A     T    103;
      =     Q   1017.3;
NETWORK
TITLE =

      A     I   1009.5;
      =     Q   1017.5;
NETWORK
TITLE =

      A     M   4711.7;
      =     Q   1017.7;
NETWORK
TITLE =

      A     I   1001.6;
      =     Q   1017.6;
NETWORK
TITLE =
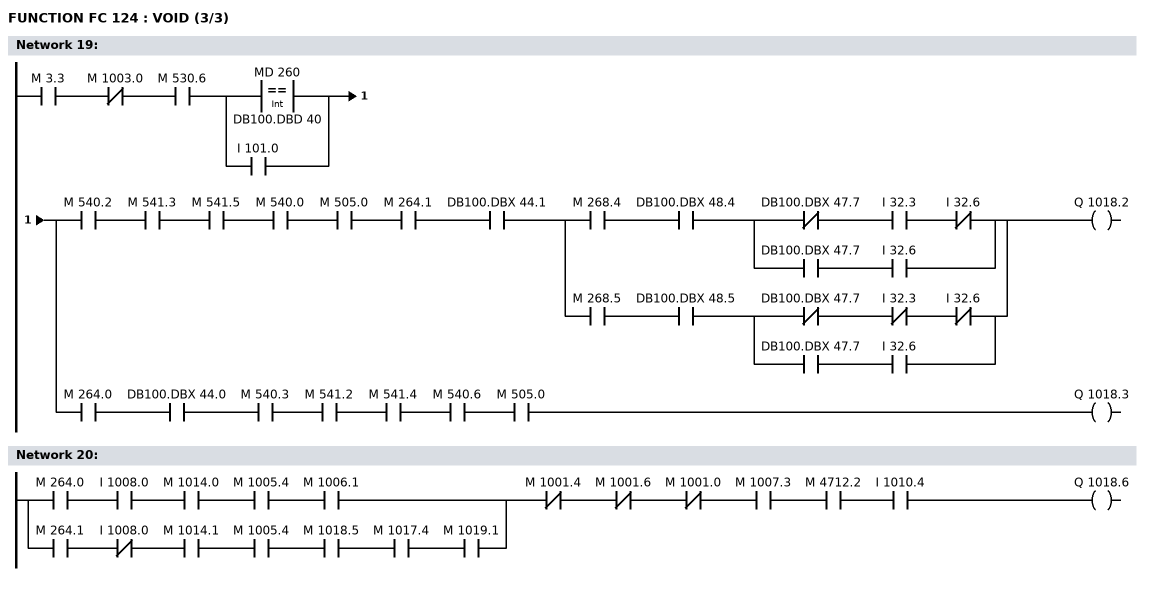

      A     M      3.3;
      AN    M   1003.0;
      A     M    530.6;
      A(    ;
      O(    ;
      L     MD   260;
      L     DB100.DBD   40;
      ==I   ;
      )     ;
      O     I    101.0;
      )     ;
      =     L      0.0;
      A     L      0.0;
      A     M    540.2;
      A     M    541.3;
      A     M    541.5;
      A     M    540.0;
      A     M    505.0;
      A     M    264.1;
      A     DB100.DBX   44.1;
      A(    ;
      A     M    268.4;
      A     DB100.DBX   48.4;
      A(    ;
      AN    DB100.DBX   47.7;
      A     I     32.3;
      AN    I     32.6;
      O     ;
      A     DB100.DBX   47.7;
      A     I     32.6;
      )     ;
      O     ;
      A     M    268.5;
      A     DB100.DBX   48.5;
      A(    ;
      AN    DB100.DBX   47.7;
      AN    I     32.3;
      AN    I     32.6;
      O     ;
      A     DB100.DBX   47.7;
      A     I     32.6;
      )     ;
      )     ;
      =     Q   1018.2;
      A     L      0.0;
      A     M    264.0;
      A     DB100.DBX   44.0;
      A     M    540.3;
      A     M    541.2;
      A     M    541.4;
      A     M    540.6;
      A     M    505.0;
      =     Q   1018.3;
NETWORK
TITLE =

      A(    ;
      A     M    264.0;
      A     I   1008.0;
      A     M   1014.0;
      A     M   1005.4;
      A     M   1006.1;
      O     ;
      A     M    264.1;
      AN    I   1008.0;
      A     M   1014.1;
      A     M   1005.4;
      A     M   1018.5;
      A     M   1017.4;
      A     M   1019.1;
      )     ;
      AN    M   1001.4;
      AN    M   1001.6;
      AN    M   1001.0;
      A     M   1007.3;
      A     M   4712.2;
      A     I   1010.4;
      =     Q   1018.6;
END_FUNCTION

FUNCTION FC 125 : VOID
TITLE =
VERSION : 0.1

BEGIN
NETWORK
TITLE =
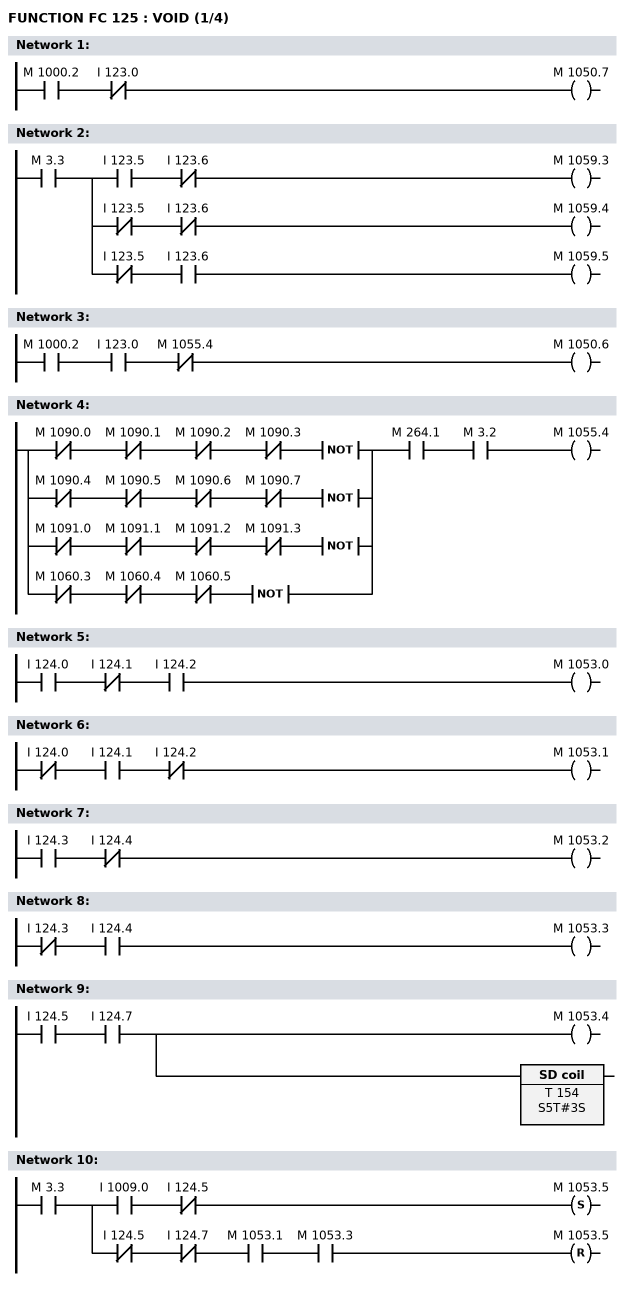

      A     M   1000.2;
      AN    I    123.0;
      =     M   1050.7;
NETWORK
TITLE =

      A     M      3.3;
      =     L      0.0;
      A     L      0.0;
      A     I    123.5;
      AN    I    123.6;
      =     M   1059.3;
      A     L      0.0;
      AN    I    123.5;
      AN    I    123.6;
      =     M   1059.4;
      A     L      0.0;
      AN    I    123.5;
      A     I    123.6;
      =     M   1059.5;
NETWORK
TITLE =

      A     M   1000.2;
      A     I    123.0;
      AN    M   1055.4;
      =     M   1050.6;
NETWORK
TITLE =

      A(    ;
      AN    M   1090.0;
      AN    M   1090.1;
      AN    M   1090.2;
      AN    M   1090.3;
      NOT   ;
      O(    ;
      AN    M   1090.4;
      AN    M   1090.5;
      AN    M   1090.6;
      AN    M   1090.7;
      NOT   ;
      )     ;
      O(    ;
      AN    M   1091.0;
      AN    M   1091.1;
      AN    M   1091.2;
      AN    M   1091.3;
      NOT   ;
      )     ;
      O(    ;
      AN    M   1060.3;
      AN    M   1060.4;
      AN    M   1060.5;
      NOT   ;
      )     ;
      )     ;
      A     M    264.1;
      A     M      3.2;
      =     M   1055.4;
NETWORK
TITLE =

      A     I    124.0;
      AN    I    124.1;
      A     I    124.2;
      =     M   1053.0;
NETWORK
TITLE =

      AN    I    124.0;
      A     I    124.1;
      AN    I    124.2;
      =     M   1053.1;
NETWORK
TITLE =

      A     I    124.3;
      AN    I    124.4;
      =     M   1053.2;
NETWORK
TITLE =

      AN    I    124.3;
      A     I    124.4;
      =     M   1053.3;
NETWORK
TITLE =

      A     I    124.5;
      A     I    124.7;
      =     M   1053.4;
      L     S5T#3S;
      SD    T    154;
NETWORK
TITLE =

      A     M      3.3;
      =     L      0.0;
      A     L      0.0;
      A     I   1009.0;
      AN    I    124.5;
      S     M   1053.5;
      A     L      0.0;
      AN    I    124.5;
      AN    I    124.7;
      A     M   1053.1;
      A     M   1053.3;
      R     M   1053.5;
NETWORK
TITLE =
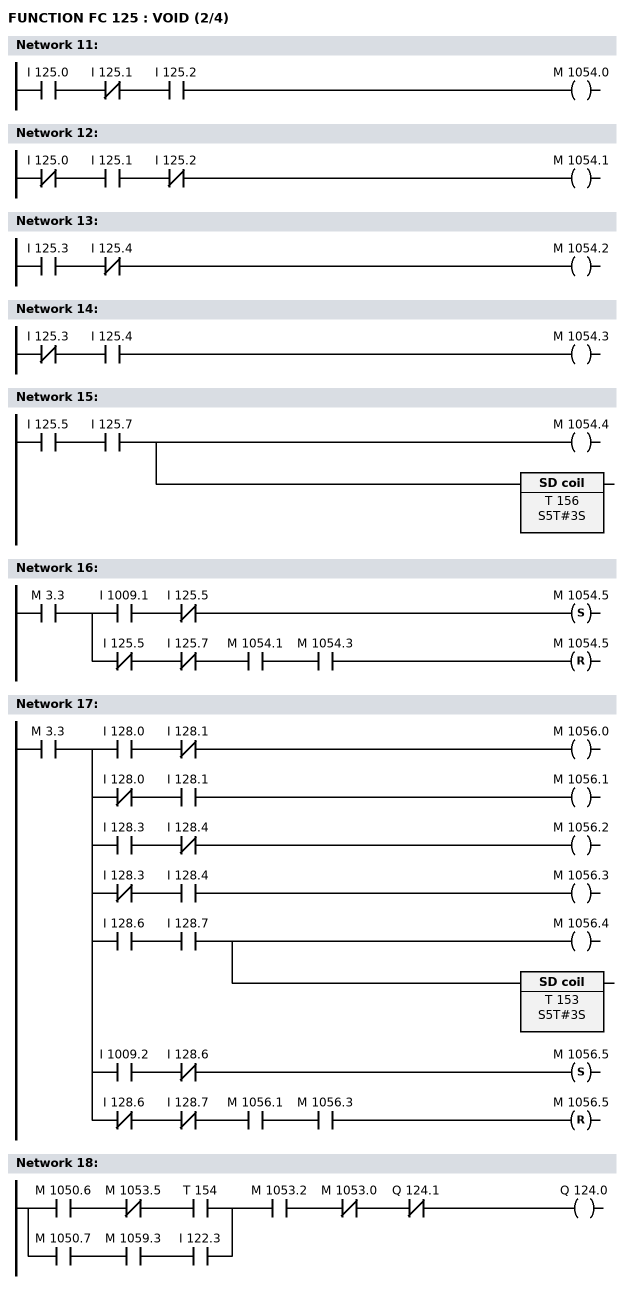

      A     I    125.0;
      AN    I    125.1;
      A     I    125.2;
      =     M   1054.0;
NETWORK
TITLE =

      AN    I    125.0;
      A     I    125.1;
      AN    I    125.2;
      =     M   1054.1;
NETWORK
TITLE =

      A     I    125.3;
      AN    I    125.4;
      =     M   1054.2;
NETWORK
TITLE =

      AN    I    125.3;
      A     I    125.4;
      =     M   1054.3;
NETWORK
TITLE =

      A     I    125.5;
      A     I    125.7;
      =     M   1054.4;
      L     S5T#3S;
      SD    T    156;
NETWORK
TITLE =

      A     M      3.3;
      =     L      0.0;
      A     L      0.0;
      A     I   1009.1;
      AN    I    125.5;
      S     M   1054.5;
      A     L      0.0;
      AN    I    125.5;
      AN    I    125.7;
      A     M   1054.1;
      A     M   1054.3;
      R     M   1054.5;
NETWORK
TITLE =

      A     M      3.3;
      =     L      0.0;
      A     L      0.0;
      A     I    128.0;
      AN    I    128.1;
      =     M   1056.0;
      A     L      0.0;
      AN    I    128.0;
      A     I    128.1;
      =     M   1056.1;
      A     L      0.0;
      A     I    128.3;
      AN    I    128.4;
      =     M   1056.2;
      A     L      0.0;
      AN    I    128.3;
      A     I    128.4;
      =     M   1056.3;
      A     L      0.0;
      A     I    128.6;
      A     I    128.7;
      =     M   1056.4;
      L     S5T#3S;
      SD    T    153;
      A     L      0.0;
      A     I   1009.2;
      AN    I    128.6;
      S     M   1056.5;
      A     L      0.0;
      AN    I    128.6;
      AN    I    128.7;
      A     M   1056.1;
      A     M   1056.3;
      R     M   1056.5;
NETWORK
TITLE =

      A(    ;
      A     M   1050.6;
      AN    M   1053.5;
      A     T    154;
      O     ;
      A     M   1050.7;
      A     M   1059.3;
      A     I    122.3;
      )     ;
      A     M   1053.2;
      AN    M   1053.0;
      AN    Q    124.1;
      =     Q    124.0;
NETWORK
TITLE =
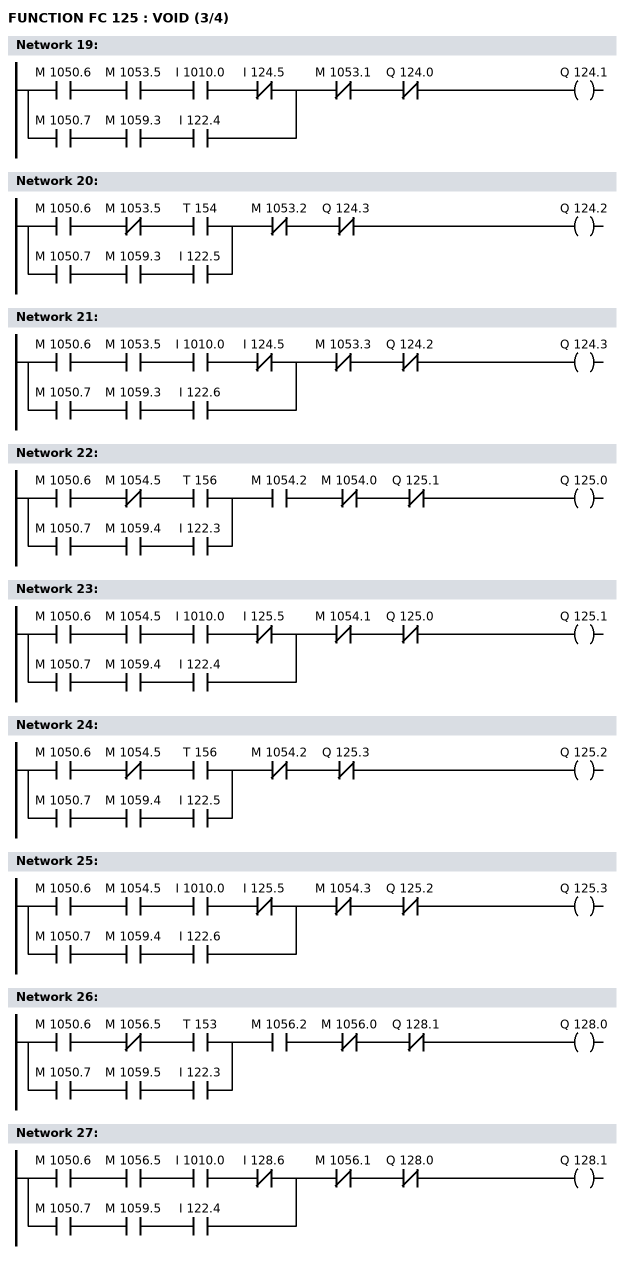

      A(    ;
      A     M   1050.6;
      A     M   1053.5;
      A     I   1010.0;
      AN    I    124.5;
      O     ;
      A     M   1050.7;
      A     M   1059.3;
      A     I    122.4;
      )     ;
      AN    M   1053.1;
      AN    Q    124.0;
      =     Q    124.1;
NETWORK
TITLE =

      A(    ;
      A     M   1050.6;
      AN    M   1053.5;
      A     T    154;
      O     ;
      A     M   1050.7;
      A     M   1059.3;
      A     I    122.5;
      )     ;
      AN    M   1053.2;
      AN    Q    124.3;
      =     Q    124.2;
NETWORK
TITLE =

      A(    ;
      A     M   1050.6;
      A     M   1053.5;
      A     I   1010.0;
      AN    I    124.5;
      O     ;
      A     M   1050.7;
      A     M   1059.3;
      A     I    122.6;
      )     ;
      AN    M   1053.3;
      AN    Q    124.2;
      =     Q    124.3;
NETWORK
TITLE =

      A(    ;
      A     M   1050.6;
      AN    M   1054.5;
      A     T    156;
      O     ;
      A     M   1050.7;
      A     M   1059.4;
      A     I    122.3;
      )     ;
      A     M   1054.2;
      AN    M   1054.0;
      AN    Q    125.1;
      =     Q    125.0;
NETWORK
TITLE =

      A(    ;
      A     M   1050.6;
      A     M   1054.5;
      A     I   1010.0;
      AN    I    125.5;
      O     ;
      A     M   1050.7;
      A     M   1059.4;
      A     I    122.4;
      )     ;
      AN    M   1054.1;
      AN    Q    125.0;
      =     Q    125.1;
NETWORK
TITLE =

      A(    ;
      A     M   1050.6;
      AN    M   1054.5;
      A     T    156;
      O     ;
      A     M   1050.7;
      A     M   1059.4;
      A     I    122.5;
      )     ;
      AN    M   1054.2;
      AN    Q    125.3;
      =     Q    125.2;
NETWORK
TITLE =

      A(    ;
      A     M   1050.6;
      A     M   1054.5;
      A     I   1010.0;
      AN    I    125.5;
      O     ;
      A     M   1050.7;
      A     M   1059.4;
      A     I    122.6;
      )     ;
      AN    M   1054.3;
      AN    Q    125.2;
      =     Q    125.3;
NETWORK
TITLE =

      A(    ;
      A     M   1050.6;
      AN    M   1056.5;
      A     T    153;
      O     ;
      A     M   1050.7;
      A     M   1059.5;
      A     I    122.3;
      )     ;
      A     M   1056.2;
      AN    M   1056.0;
      AN    Q    128.1;
      =     Q    128.0;
NETWORK
TITLE =

      A(    ;
      A     M   1050.6;
      A     M   1056.5;
      A     I   1010.0;
      AN    I    128.6;
      O     ;
      A     M   1050.7;
      A     M   1059.5;
      A     I    122.4;
      )     ;
      AN    M   1056.1;
      AN    Q    128.0;
      =     Q    128.1;
NETWORK
TITLE =
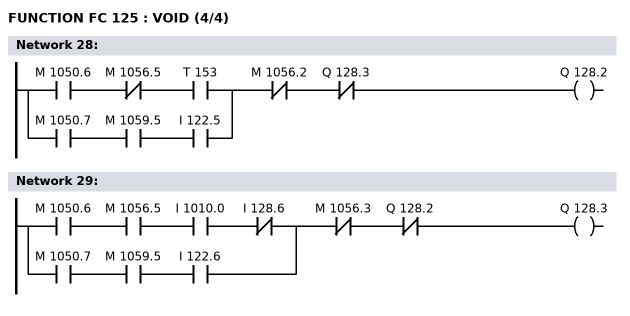

      A(    ;
      A     M   1050.6;
      AN    M   1056.5;
      A     T    153;
      O     ;
      A     M   1050.7;
      A     M   1059.5;
      A     I    122.5;
      )     ;
      AN    M   1056.2;
      AN    Q    128.3;
      =     Q    128.2;
NETWORK
TITLE =

      A(    ;
      A     M   1050.6;
      A     M   1056.5;
      A     I   1010.0;
      AN    I    128.6;
      O     ;
      A     M   1050.7;
      A     M   1059.5;
      A     I    122.6;
      )     ;
      AN    M   1056.3;
      AN    Q    128.2;
      =     Q    128.3;
END_FUNCTION

FUNCTION FC 126 : VOID
TITLE =
VERSION : 0.1

BEGIN
NETWORK
TITLE =
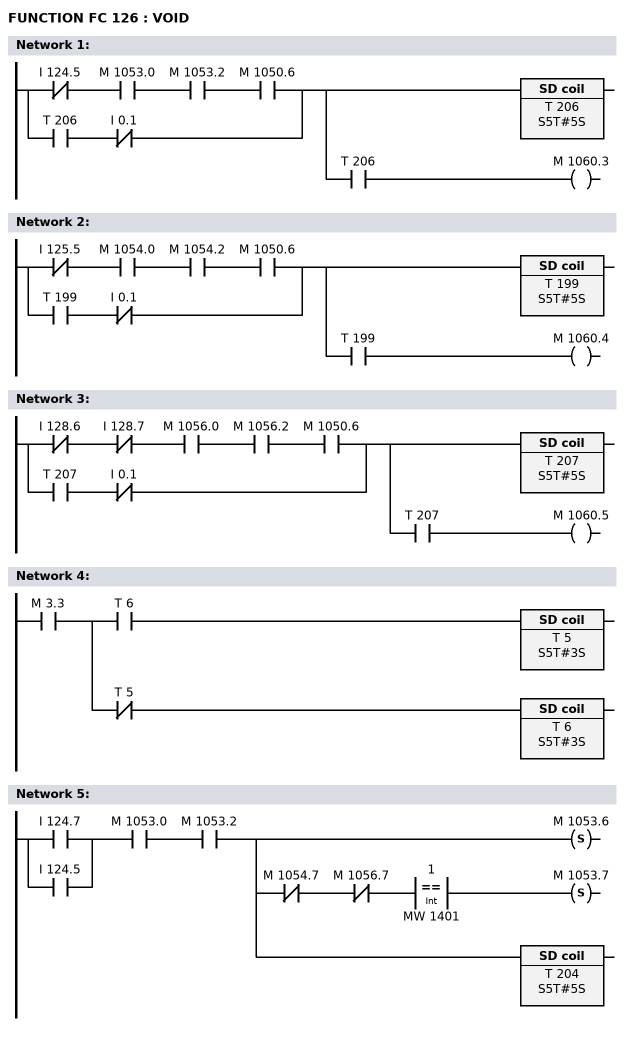

      AN    I    124.5;
      A     M   1053.0;
      A     M   1053.2;
      A     M   1050.6;
      O     ;
      A     T    206;
      AN    I      0.1;
      =     L      0.0;
      A     L      0.0;
      BLD   102;
      L     S5T#5S;
      SD    T    206;
      A     L      0.0;
      A     T    206;
      =     M   1060.3;
NETWORK
TITLE =

      AN    I    125.5;
      A     M   1054.0;
      A     M   1054.2;
      A     M   1050.6;
      O     ;
      A     T    199;
      AN    I      0.1;
      =     L      0.0;
      A     L      0.0;
      BLD   102;
      L     S5T#5S;
      SD    T    199;
      A     L      0.0;
      A     T    199;
      =     M   1060.4;
NETWORK
TITLE =

      AN    I    128.6;
      AN    I    128.7;
      A     M   1056.0;
      A     M   1056.2;
      A     M   1050.6;
      O     ;
      A     T    207;
      AN    I      0.1;
      =     L      0.0;
      A     L      0.0;
      BLD   102;
      L     S5T#5S;
      SD    T    207;
      A     L      0.0;
      A     T    207;
      =     M   1060.5;
NETWORK
TITLE =

      A     M      3.3;
      =     L      0.0;
      A     L      0.0;
      A     T      6;
      L     S5T#3S;
      SD    T      5;
      A     L      0.0;
      AN    T      5;
      L     S5T#3S;
      SD    T      6;
NETWORK
TITLE =

      A(    ;
      O     I    124.7;
      O     I    124.5;
      )     ;
      A     M   1053.0;
      A     M   1053.2;
      =     L      0.0;
      A     L      0.0;
      BLD   102;
      S     M   1053.6;
      A     L      0.0;
      AN    M   1054.7;
      AN    M   1056.7;
      A(    ;
      L     1;
      L     MW  1401;
      ==I   ;
      )     ;
      S     M   1053.7;
      A     L      0.0;
      BLD   102;
      L     S5T#5S;
      SD    T    204;
NETWORK
TITLE =

      ON    I    124.5;
      ON    I    124.7;
      ON    M   1053.0;
      O     I    122.1;
      =     L      0.0;
      A     L      0.0;
      A     T    205;
      =     L      0.1;
      A     L      0.1;
      BLD   102;
      R     M   1053.6;
      A     L      0.1;
      A     I   1009.0;
      R     M   1053.7;
      A(    ;
      A     L      0.1;
      A(    ;
      L     0;
      L     MW  1401;
      <>I   ;
      )     ;
      JNB   _001;
      L     MW  1401;
      T     MW  1421;
      SET   ;
      SAVE  ;
      CLR   ;
_001: A     BR;
      )     ;
      JNB   _002;
      L     0;
      T     MW  1401;
_002: NOP   0;
      A     L      0.0;
      BLD   102;
      L     S5T#3S;
      SD    T    205;
NETWORK
TITLE =
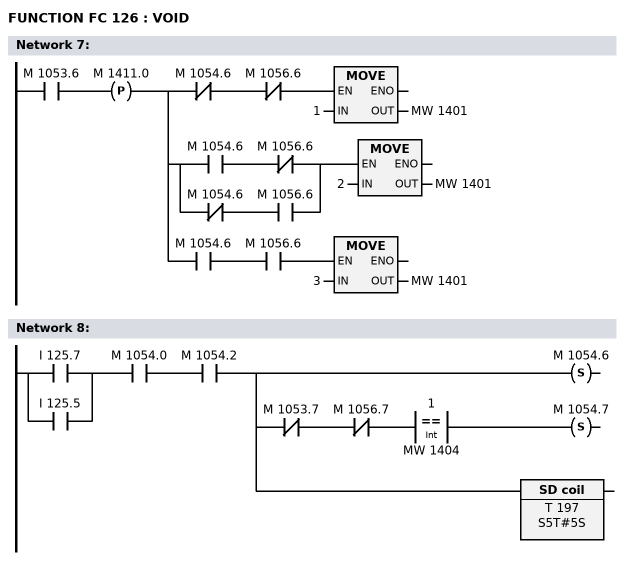

      A     M   1053.6;
      FP    M   1411.0;
      =     L      0.0;
      A     L      0.0;
      AN    M   1054.6;
      AN    M   1056.6;
      JNB   _003;
      L     1;
      T     MW  1401;
_003: NOP   0;
      A     L      0.0;
      A(    ;
      A     M   1054.6;
      AN    M   1056.6;
      O     ;
      AN    M   1054.6;
      A     M   1056.6;
      )     ;
      JNB   _004;
      L     2;
      T     MW  1401;
_004: NOP   0;
      A     L      0.0;
      A     M   1054.6;
      A     M   1056.6;
      JNB   _005;
      L     3;
      T     MW  1401;
_005: NOP   0;
NETWORK
TITLE =

      A(    ;
      O     I    125.7;
      O     I    125.5;
      )     ;
      A     M   1054.0;
      A     M   1054.2;
      =     L      0.0;
      A     L      0.0;
      BLD   102;
      S     M   1054.6;
      A     L      0.0;
      AN    M   1053.7;
      AN    M   1056.7;
      A(    ;
      L     1;
      L     MW  1404;
      ==I   ;
      )     ;
      S     M   1054.7;
      A     L      0.0;
      BLD   102;
      L     S5T#5S;
      SD    T    197;
NETWORK
TITLE =

      ON    I    125.5;
      ON    I    125.7;
      ON    M   1054.0;
      O     I    122.1;
      =     L      0.0;
      A     L      0.0;
      A     T    198;
      =     L      0.1;
      A     L      0.1;
      BLD   102;
      R     M   1054.6;
      A     L      0.1;
      A     I   1009.1;
      R     M   1054.7;
      A(    ;
      A     L      0.1;
      A(    ;
      L     0;
      L     MW  1404;
      <>I   ;
      )     ;
      JNB   _006;
      L     MW  1404;
      T     MW  1424;
      SET   ;
      SAVE  ;
      CLR   ;
_006: A     BR;
      )     ;
      JNB   _007;
      L     0;
      T     MW  1404;
_007: NOP   0;
      A     L      0.0;
      BLD   102;
      L     S5T#3S;
      SD    T    198;
NETWORK
TITLE =
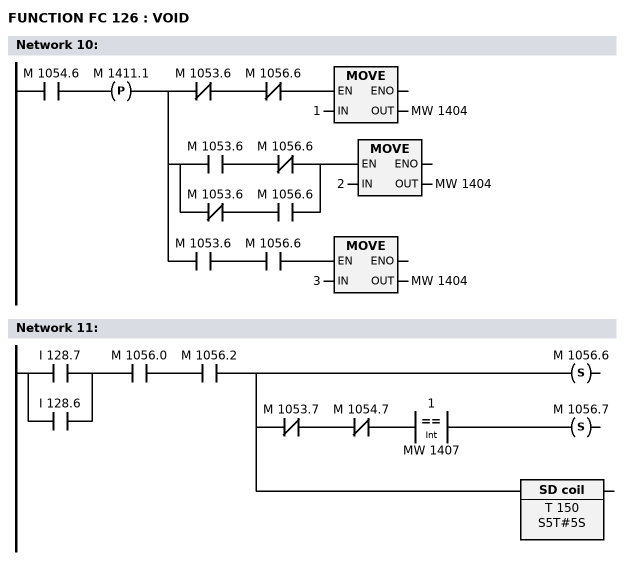

      A     M   1054.6;
      FP    M   1411.1;
      =     L      0.0;
      A     L      0.0;
      AN    M   1053.6;
      AN    M   1056.6;
      JNB   _008;
      L     1;
      T     MW  1404;
_008: NOP   0;
      A     L      0.0;
      A(    ;
      A     M   1053.6;
      AN    M   1056.6;
      O     ;
      AN    M   1053.6;
      A     M   1056.6;
      )     ;
      JNB   _009;
      L     2;
      T     MW  1404;
_009: NOP   0;
      A     L      0.0;
      A     M   1053.6;
      A     M   1056.6;
      JNB   _00a;
      L     3;
      T     MW  1404;
_00a: NOP   0;
NETWORK
TITLE =

      A(    ;
      O     I    128.7;
      O     I    128.6;
      )     ;
      A     M   1056.0;
      A     M   1056.2;
      =     L      0.0;
      A     L      0.0;
      BLD   102;
      S     M   1056.6;
      A     L      0.0;
      AN    M   1053.7;
      AN    M   1054.7;
      A(    ;
      L     1;
      L     MW  1407;
      ==I   ;
      )     ;
      S     M   1056.7;
      A     L      0.0;
      BLD   102;
      L     S5T#5S;
      SD    T    150;
NETWORK
TITLE =

      ON    I    128.6;
      ON    I    128.7;
      ON    M   1056.0;
      O     I    122.1;
      =     L      0.0;
      A     L      0.0;
      A     T    151;
      =     L      0.1;
      A     L      0.1;
      BLD   102;
      R     M   1056.6;
      A     L      0.1;
      A     I   1009.2;
      R     M   1056.7;
      A(    ;
      A     L      0.1;
      A(    ;
      L     0;
      L     MW  1407;
      <>I   ;
      )     ;
      JNB   _00b;
      L     MW  1407;
      T     MW  1427;
      SET   ;
      SAVE  ;
      CLR   ;
_00b: A     BR;
      )     ;
      JNB   _00c;
      L     0;
      T     MW  1407;
_00c: NOP   0;
      A     L      0.0;
      BLD   102;
      L     S5T#3S;
      SD    T    151;
NETWORK
TITLE =
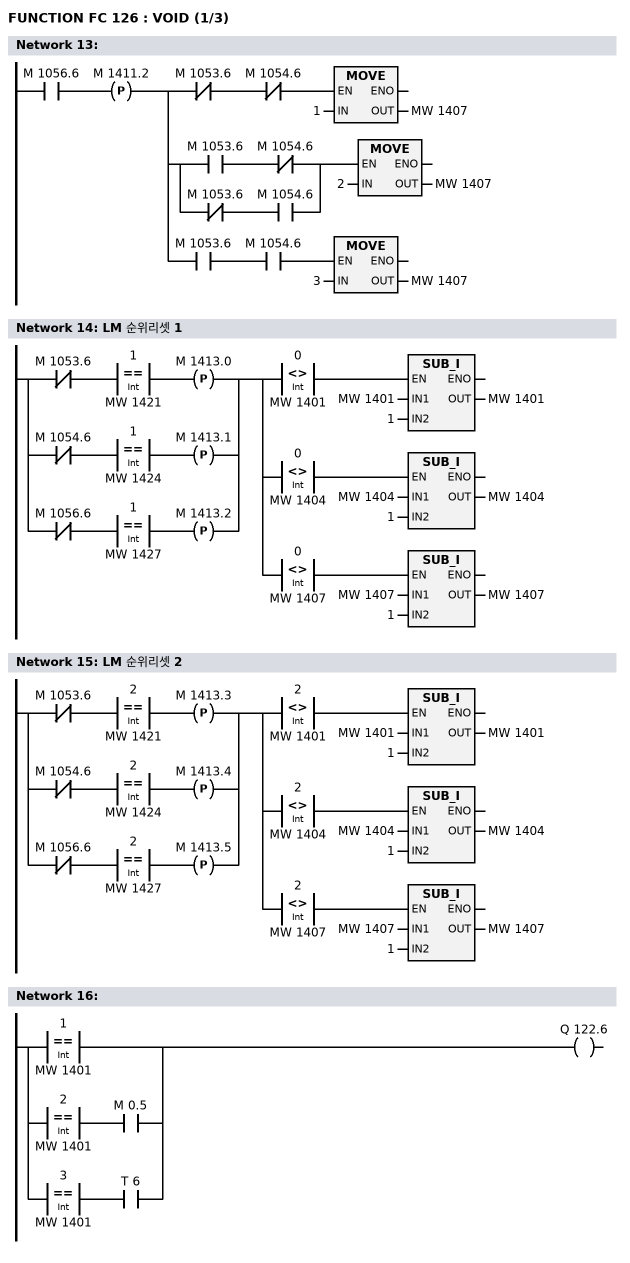

      A     M   1056.6;
      FP    M   1411.2;
      =     L      0.0;
      A     L      0.0;
      AN    M   1053.6;
      AN    M   1054.6;
      JNB   _00d;
      L     1;
      T     MW  1407;
_00d: NOP   0;
      A     L      0.0;
      A(    ;
      A     M   1053.6;
      AN    M   1054.6;
      O     ;
      AN    M   1053.6;
      A     M   1054.6;
      )     ;
      JNB   _00e;
      L     2;
      T     MW  1407;
_00e: NOP   0;
      A     L      0.0;
      A     M   1053.6;
      A     M   1054.6;
      JNB   _00f;
      L     3;
      T     MW  1407;
_00f: NOP   0;
NETWORK
TITLE =LM 순위리셋 1

      AN    M   1053.6;
      A(    ;
      L     1;
      L     MW  1421;
      ==I   ;
      )     ;
      FP    M   1413.0;
      O(    ;
      AN    M   1054.6;
      A(    ;
      L     1;
      L     MW  1424;
      ==I   ;
      )     ;
      FP    M   1413.1;
      )     ;
      O(    ;
      AN    M   1056.6;
      A(    ;
      L     1;
      L     MW  1427;
      ==I   ;
      )     ;
      FP    M   1413.2;
      )     ;
      =     L      0.0;
      A     L      0.0;
      A(    ;
      L     0;
      L     MW  1401;
      <>I   ;
      )     ;
      JNB   _010;
      L     MW  1401;
      L     1;
      -I    ;
      T     MW  1401;
_010: NOP   0;
      A     L      0.0;
      A(    ;
      L     0;
      L     MW  1404;
      <>I   ;
      )     ;
      JNB   _011;
      L     MW  1404;
      L     1;
      -I    ;
      T     MW  1404;
_011: NOP   0;
      A     L      0.0;
      A(    ;
      L     0;
      L     MW  1407;
      <>I   ;
      )     ;
      JNB   _012;
      L     MW  1407;
      L     1;
      -I    ;
      T     MW  1407;
_012: NOP   0;
NETWORK
TITLE =LM 순위리셋 2

      AN    M   1053.6;
      A(    ;
      L     2;
      L     MW  1421;
      ==I   ;
      )     ;
      FP    M   1413.3;
      O(    ;
      AN    M   1054.6;
      A(    ;
      L     2;
      L     MW  1424;
      ==I   ;
      )     ;
      FP    M   1413.4;
      )     ;
      O(    ;
      AN    M   1056.6;
      A(    ;
      L     2;
      L     MW  1427;
      ==I   ;
      )     ;
      FP    M   1413.5;
      )     ;
      =     L      0.0;
      A     L      0.0;
      A(    ;
      L     2;
      L     MW  1401;
      <>I   ;
      )     ;
      JNB   _013;
      L     MW  1401;
      L     1;
      -I    ;
      T     MW  1401;
_013: NOP   0;
      A     L      0.0;
      A(    ;
      L     2;
      L     MW  1404;
      <>I   ;
      )     ;
      JNB   _014;
      L     MW  1404;
      L     1;
      -I    ;
      T     MW  1404;
_014: NOP   0;
      A     L      0.0;
      A(    ;
      L     2;
      L     MW  1407;
      <>I   ;
      )     ;
      JNB   _015;
      L     MW  1407;
      L     1;
      -I    ;
      T     MW  1407;
_015: NOP   0;
NETWORK
TITLE =

      O(    ;
      L     1;
      L     MW  1401;
      ==I   ;
      )     ;
      O     ;
      A(    ;
      L     2;
      L     MW  1401;
      ==I   ;
      )     ;
      A     M      0.5;
      O     ;
      A(    ;
      L     3;
      L     MW  1401;
      ==I   ;
      )     ;
      A     T      6;
      =     Q    122.6;
NETWORK
TITLE =
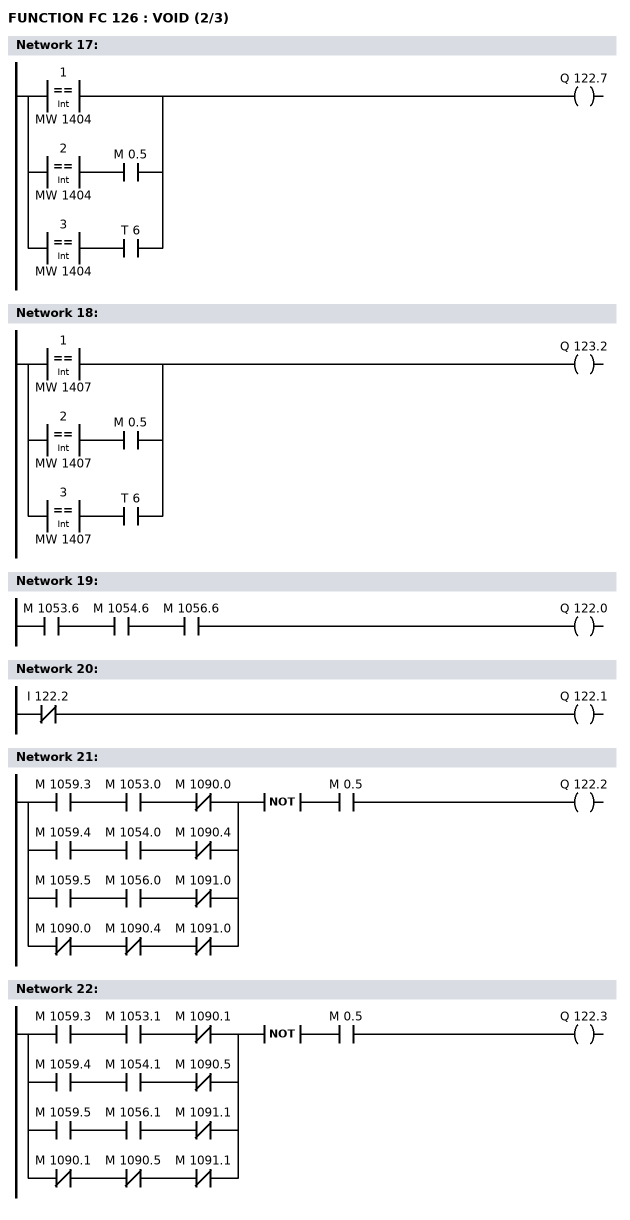

      O(    ;
      L     1;
      L     MW  1404;
      ==I   ;
      )     ;
      O     ;
      A(    ;
      L     2;
      L     MW  1404;
      ==I   ;
      )     ;
      A     M      0.5;
      O     ;
      A(    ;
      L     3;
      L     MW  1404;
      ==I   ;
      )     ;
      A     T      6;
      =     Q    122.7;
NETWORK
TITLE =

      O(    ;
      L     1;
      L     MW  1407;
      ==I   ;
      )     ;
      O     ;
      A(    ;
      L     2;
      L     MW  1407;
      ==I   ;
      )     ;
      A     M      0.5;
      O     ;
      A(    ;
      L     3;
      L     MW  1407;
      ==I   ;
      )     ;
      A     T      6;
      =     Q    123.2;
NETWORK
TITLE =

      A     M   1053.6;
      A     M   1054.6;
      A     M   1056.6;
      =     Q    122.0;
NETWORK
TITLE =

      AN    I    122.2;
      =     Q    122.1;
NETWORK
TITLE =

      A     M   1059.3;
      A     M   1053.0;
      AN    M   1090.0;
      O     ;
      A     M   1059.4;
      A     M   1054.0;
      AN    M   1090.4;
      O     ;
      A     M   1059.5;
      A     M   1056.0;
      AN    M   1091.0;
      O     ;
      AN    M   1090.0;
      AN    M   1090.4;
      AN    M   1091.0;
      NOT   ;
      A     M      0.5;
      =     Q    122.2;
NETWORK
TITLE =

      A     M   1059.3;
      A     M   1053.1;
      AN    M   1090.1;
      O     ;
      A     M   1059.4;
      A     M   1054.1;
      AN    M   1090.5;
      O     ;
      A     M   1059.5;
      A     M   1056.1;
      AN    M   1091.1;
      O     ;
      AN    M   1090.1;
      AN    M   1090.5;
      AN    M   1091.1;
      NOT   ;
      A     M      0.5;
      =     Q    122.3;
NETWORK
TITLE =
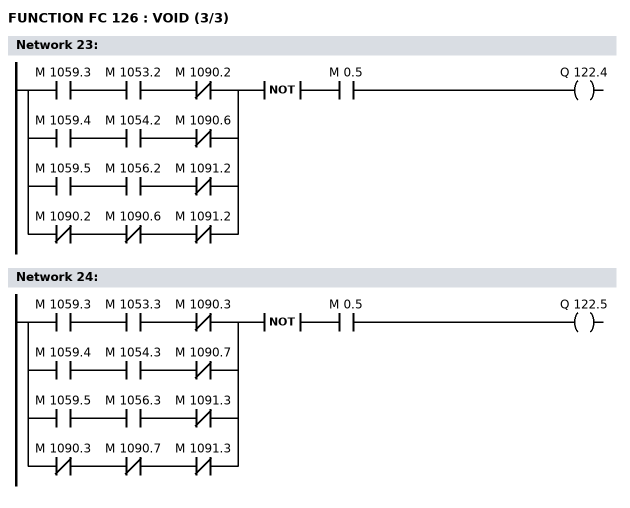

      A     M   1059.3;
      A     M   1053.2;
      AN    M   1090.2;
      O     ;
      A     M   1059.4;
      A     M   1054.2;
      AN    M   1090.6;
      O     ;
      A     M   1059.5;
      A     M   1056.2;
      AN    M   1091.2;
      O     ;
      AN    M   1090.2;
      AN    M   1090.6;
      AN    M   1091.2;
      NOT   ;
      A     M      0.5;
      =     Q    122.4;
NETWORK
TITLE =

      A     M   1059.3;
      A     M   1053.3;
      AN    M   1090.3;
      O     ;
      A     M   1059.4;
      A     M   1054.3;
      AN    M   1090.7;
      O     ;
      A     M   1059.5;
      A     M   1056.3;
      AN    M   1091.3;
      O     ;
      AN    M   1090.3;
      AN    M   1090.7;
      AN    M   1091.3;
      NOT   ;
      A     M      0.5;
      =     Q    122.5;
END_FUNCTION

FUNCTION FC 324 : VOID
TITLE =
VERSION : 0.1

BEGIN
NETWORK
TITLE =DP DIAGNOSTIC FOR DP MASTER SYSTEM(1)

      AN    OV;
      =     L      0.0;
      BLD   103;
      A     OV;
      =     L      0.1;
      BLD   103;
      CALL FC   325 (
           CHECK_ACTIV              := L      0.0,
           EXTERNAL_DP_INTERFACE    := L      0.1,
           DP_MASTERSYSTEM          := 1,
           DATA_FIELD               := P#DB325.DBX0.0 BYTE 50,
           SUM_SLAVES_DIAG          := DB325.DBW   82,
           LIST_SLAVES_NOT_PRESENT  := P#DB325.DBX 50.0 DWORD 4,
           LIST_SLAVES_ERROR        := P#DB325.DBX 66.0 DWORD 4,
           RETVAL                   := DB325.DBW   84,
           BUSY                     := DB325.DBX   90.0);
      NOP   0;
NETWORK
TITLE =
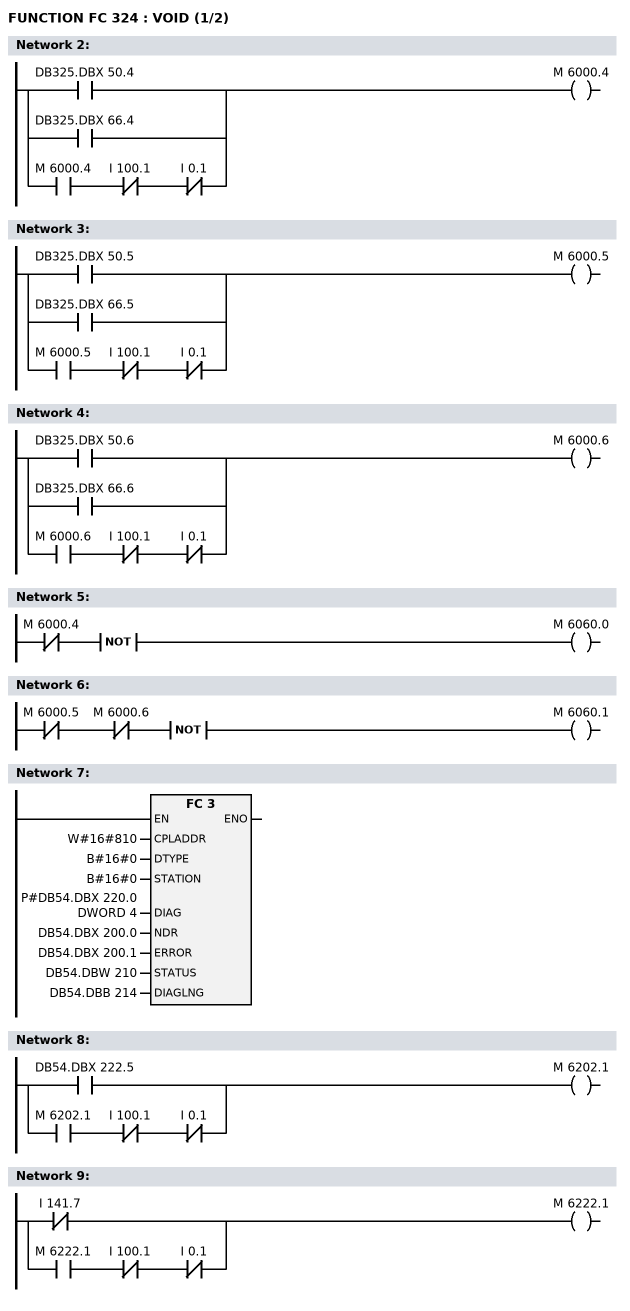

      O     DB325.DBX   50.4;
      O     DB325.DBX   66.4;
      O     ;
      A     M   6000.4;
      AN    I    100.1;
      AN    I      0.1;
      =     M   6000.4;
NETWORK
TITLE =

      O     DB325.DBX   50.5;
      O     DB325.DBX   66.5;
      O     ;
      A     M   6000.5;
      AN    I    100.1;
      AN    I      0.1;
      =     M   6000.5;
NETWORK
TITLE =

      O     DB325.DBX   50.6;
      O     DB325.DBX   66.6;
      O     ;
      A     M   6000.6;
      AN    I    100.1;
      AN    I      0.1;
      =     M   6000.6;
NETWORK
TITLE =

      AN    M   6000.4;
      NOT   ;
      =     M   6060.0;
NETWORK
TITLE =

      AN    M   6000.5;
      AN    M   6000.6;
      NOT   ;
      =     M   6060.1;
NETWORK
TITLE =

      CALL FC     3 (
           CPLADDR                  := W#16#810,
           DTYPE                    := B#16#0,
           STATION                  := B#16#0,
           DIAG                     := P#DB54.DBX 220.0 DWORD 4,
           NDR                      := DB54.DBX  200.0,
           ERROR                    := DB54.DBX  200.1,
           STATUS                   := DB54.DBW  210,
           DIAGLNG                  := DB54.DBB  214);
      NOP   0;
NETWORK
TITLE =

      O     DB54.DBX  222.5;
      O     ;
      A     M   6202.1;
      AN    I    100.1;
      AN    I      0.1;
      =     M   6202.1;
NETWORK
TITLE =

      ON    I    141.7;
      O     ;
      A     M   6222.1;
      AN    I    100.1;
      AN    I      0.1;
      =     M   6222.1;
NETWORK
TITLE =
